LIN {X 0,Y 305.638,Z 167.911,A -85,B 0,C 180,E1 -15829.4,E2 -15829.4} C_VEL
LIN {X 0,Y 305.807,Z 167.885,A -85,B 0,C 180,E1 -15832.074,E2 -15832.074} C_VEL
LIN {X 0,Y 305.686,Z 167.907,A -85,B 0,C 180,E1 -15834.723,E2 -15834.723} C_VEL
LIN {X 0,Y 305.955,Z 167.869,A -85,B 0,C 180,E1 -15838.684,E2 -15838.684} C_VEL
LIN {X 0,Y 305.957,Z 167.872,A -85,B 0,C 180,E1 -15841.316,E2 -15841.316} C_VEL
LIN {X 0,Y 305.845,Z 167.883,A -85,B 0,C 180,E1 -15846.598,E2 -15846.598} C_VEL
LIN {X 0,Y 305.735,Z 167.899,A -85,B 0,C 180,E1 -15849.26,E2 -15849.26} C_VEL
LIN {X 0,Y 305.588,Z 167.911,A -85,B 0,C 180,E1 -15853.296,E2 -15853.296} C_VEL
LIN {X 0,Y 305.593,Z 167.918,A -85,B 0,C 180,E1 -15856.02,E2 -15856.02} C_VEL
LIN {X 0,Y 305.56,Z 167.916,A -85,B 0,C 180,E1 -15859.436,E2 -15859.436} C_VEL
LIN {X 0,Y 305.485,Z 167.93,A -85,B 0,C 180,E1 -15863.039,E2 -15863.039} C_VEL
LIN {X 0,Y 305.546,Z 167.925,A -85,B 0,C 180,E1 -15866.227,E2 -15866.227} C_VEL
LIN {X 0,Y 305.487,Z 167.929,A -85,B 0,C 180,E1 -15869.047,E2 -15869.047} C_VEL
LIN {X 0,Y 305.443,Z 167.94,A -85,B 0,C 180,E1 -15871.952,E2 -15871.952} C_VEL
LIN {X 0,Y 305.462,Z 167.931,A -85,B 0,C 180,E1 -15875.113,E2 -15875.113} C_VEL
LIN {X 0,Y 305.439,Z 167.934,A -85,B 0,C 180,E1 -15878.527,E2 -15878.527} C_VEL
LIN {X 0,Y 305.454,Z 167.934,A -85,B 0,C 180,E1 -15882.586,E2 -15882.586} C_VEL
LIN {X 0,Y 305.421,Z 167.938,A -85,B 0,C 180,E1 -15886.344,E2 -15886.344} C_VEL
LIN {X 0,Y 305.409,Z 167.941,A -85,B 0,C 180,E1 -15889.885,E2 -15889.885} C_VEL
LIN {X 0,Y 305.479,Z 167.934,A -85,B 0,C 180,E1 -15893.633,E2 -15893.633} C_VEL
LIN {X 0,Y 305.508,Z 167.974,A -85,B 0,C 180,E1 -15896.982,E2 -15896.982} C_VEL
LIN {X 0,Y 307.705,Z 177.752,A -85,B 0,C 180,E1 -15900.218,E2 -15900.218} C_VEL
LIN {X 0,Y 309.879,Z 188.802,A -85,B 0,C 180,E1 -15903.685,E2 -15903.685} C_VEL
LIN {X 0,Y 311.303,Z 192.906,A -85,B 0,C 180,E1 -15903.964,E2 -15903.964} C_VEL
LIN {X 0,Y 315.786,Z 216.896,A -85,B 0,C 180,E1 -15904.949,E2 -15904.949} C_VEL
LIN {X 0,Y 317.76,Z 229.786,A -85,B 0,C 180,E1 -15905.428,E2 -15905.428} C_VEL
LIN {X 0,Y 316.105,Z 297.454,A -85,B 0,C 180,E1 -15906.973,E2 -15906.973} C_VEL
LIN {X 0,Y 315.2,Z 310.618,A -85,B 0,C 180,E1 -15907.51,E2 -15907.51} C_VEL
LIN {X 0,Y 314.151,Z 322.724,A -85,B 0,C 180,E1 -15908.252,E2 -15908.252} C_VEL
LIN {X 0,Y 312.759,Z 334.943,A -85,B 0,C 180,E1 -15909.273,E2 -15909.273} C_VEL
LIN {X 0,Y 311.132,Z 346.512,A -85,B 0,C 180,E1 -15910.538,E2 -15910.538} C_VEL
LIN {X 0,Y 309.594,Z 356.932,A -85,B 0,C 180,E1 -15911.983,E2 -15911.983} C_VEL
LIN {X 0,Y 308.215,Z 366.424,A -85,B 0,C 180,E1 -15913.633,E2 -15913.633} C_VEL
LIN {X 0,Y 306.873,Z 374.691,A -85,B 0,C 180,E1 -15915.409,E2 -15915.409} C_VEL
LIN {X 0,Y 305.599,Z 382.114,A -85,B 0,C 180,E1 -15917.381,E2 -15917.381} C_VEL
LIN {X 0,Y 304.716,Z 388.078,A -85,B 0,C 180,E1 -15919.367,E2 -15919.367} C_VEL
LIN {X 0,Y 304.12,Z 392.792,A -85,B 0,C 180,E1 -15921.361,E2 -15921.361} C_VEL
LIN {X 0,Y 303.74,Z 396.394,A -85,B 0,C 180,E1 -15923.357,E2 -15923.357} C_VEL
LIN {X 0,Y 303.618,Z 398.252,A -85,B 0,C 180,E1 -15924.687,E2 -15924.687} C_VEL
LIN {X 0,Y 303.587,Z 399.647,A -85,B 0,C 180,E1 -15926.018,E2 -15926.018} C_VEL
LIN {X 0,Y 303.598,Z 400.642,A -85,B 0,C 180,E1 -15927.346,E2 -15927.346} C_VEL
LIN {X 0,Y 303.556,Z 401.248,A -85,B 0,C 180,E1 -15928.673,E2 -15928.673} C_VEL
LIN {X 0,Y 303.565,Z 401.461,A -85,B 0,C 180,E1 -15930,E2 -15930} C_VEL
LIN {X 0,Y 303.556,Z 401.24,A -85,B 0,C 180,E1 -15931.327,E2 -15931.327} C_VEL
LIN {X 0,Y 303.598,Z 400.63,A -85,B 0,C 180,E1 -15932.654,E2 -15932.654} C_VEL
LIN {X 0,Y 303.588,Z 399.63,A -85,B 0,C 180,E1 -15933.982,E2 -15933.982} C_VEL
LIN {X 0,Y 303.618,Z 397.941,A -85,B 0,C 180,E1 -15935.53,E2 -15935.53} C_VEL
LIN {X 0,Y 303.958,Z 394.057,A -85,B 0,C 180,E1 -15937.974,E2 -15937.974} C_VEL
LIN {X 0,Y 304.472,Z 389.713,A -85,B 0,C 180,E1 -15939.969,E2 -15939.969} C_VEL
LIN {X 0,Y 305.231,Z 384.18,A -85,B 0,C 180,E1 -15941.96,E2 -15941.96} C_VEL
LIN {X 0,Y 306.397,Z 377.279,A -85,B 0,C 180,E1 -15943.936,E2 -15943.936} C_VEL
LIN {X 0,Y 307.521,Z 370.231,A -85,B 0,C 180,E1 -15945.577,E2 -15945.577} C_VEL
LIN {X 0,Y 308.797,Z 361.735,A -85,B 0,C 180,E1 -15947.21,E2 -15947.21} C_VEL
LIN {X 0,Y 310.369,Z 351.24,A -85,B 0,C 180,E1 -15948.825,E2 -15948.825} C_VEL
LIN {X 0,Y 312.149,Z 339.43,A -85,B 0,C 180,E1 -15950.253,E2 -15950.253} C_VEL
LIN {X 0,Y 313.536,Z 327.532,A -85,B 0,C 180,E1 -15951.361,E2 -15951.361} C_VEL
LIN {X 0,Y 314.818,Z 315.152,A -85,B 0,C 180,E1 -15952.217,E2 -15952.217} C_VEL
LIN {X 0,Y 315.848,Z 302.407,A -85,B 0,C 180,E1 -15952.83,E2 -15952.83} C_VEL
LIN {X 0,Y 316.401,Z 288.944,A -85,B 0,C 180,E1 -15953.22,E2 -15953.22} C_VEL
LIN {X 0,Y 317.6,Z 229.007,A -85,B 0,C 180,E1 -15954.578,E2 -15954.578} C_VEL
LIN {X 0,Y 313.198,Z 202.348,A -85,B 0,C 180,E1 -15955.605,E2 -15955.605} C_VEL
LIN {X 0,Y 311.081,Z 192.208,A -85,B 0,C 180,E1 -15956.045,E2 -15956.045} C_VEL
LIN {X 0,Y 309.905,Z 188.891,A -85,B 0,C 180,E1 -15956.258,E2 -15956.258} C_VEL
LIN {X 0,Y 307.676,Z 177.689,A -85,B 0,C 180,E1 -15959.772,E2 -15959.772} C_VEL
LIN {X 0,Y 305.494,Z 167.931,A -85,B 0,C 180,E1 -15963.02,E2 -15963.02} C_VEL
LIN {X 0,Y 305.469,Z 167.937,A -85,B 0,C 180,E1 -15966.74,E2 -15966.74} C_VEL
LIN {X 0,Y 305.409,Z 167.944,A -85,B 0,C 180,E1 -15970.59,E2 -15970.59} C_VEL
LIN {X 0,Y 305.421,Z 167.939,A -85,B 0,C 180,E1 -15973.656,E2 -15973.656} C_VEL
LIN {X 0,Y 305.454,Z 167.934,A -85,B 0,C 180,E1 -15977.414,E2 -15977.414} C_VEL
LIN {X 0,Y 305.467,Z 167.933,A -85,B 0,C 180,E1 -15981.596,E2 -15981.596} C_VEL
LIN {X 0,Y 305.462,Z 167.934,A -85,B 0,C 180,E1 -15984.887,E2 -15984.887} C_VEL
LIN {X 0,Y 305.441,Z 167.939,A -85,B 0,C 180,E1 -15988.358,E2 -15988.358} C_VEL
LIN {X 0,Y 305.486,Z 167.93,A -85,B 0,C 180,E1 -15991.11,E2 -15991.11} C_VEL
LIN {X 0,Y 305.505,Z 167.932,A -85,B 0,C 180,E1 -15994.082,E2 -15994.082} C_VEL
LIN {X 0,Y 305.481,Z 167.931,A -85,B 0,C 180,E1 -15998.401,E2 -15998.401} C_VEL
LIN {X 0,Y 305.579,Z 167.919,A -85,B 0,C 180,E1 -16001.217,E2 -16001.217} C_VEL
LIN {X 0,Y 305.649,Z 167.912,A -85,B 0,C 180,E1 -16005.349,E2 -16005.349} C_VEL
LIN {X 0,Y 305.635,Z 167.913,A -85,B 0,C 180,E1 -16009.4,E2 -16009.4} C_VEL
LIN {X 0,Y 305.796,Z 167.89,A -85,B 0,C 180,E1 -16012.074,E2 -16012.074} C_VEL
LIN {X 0,Y 305.686,Z 167.903,A -85,B 0,C 180,E1 -16014.723,E2 -16014.723} C_VEL
LIN {X 0,Y 305.957,Z 167.87,A -85,B 0,C 180,E1 -16018.684,E2 -16018.684} C_VEL
LIN {X 0,Y 305.956,Z 167.875,A -85,B 0,C 180,E1 -16021.316,E2 -16021.316} C_VEL
LIN {X 0,Y 305.683,Z 167.904,A -85,B 0,C 180,E1 -16025.277,E2 -16025.277} C_VEL
LIN {X 0,Y 305.8,Z 167.891,A -85,B 0,C 180,E1 -16027.926,E2 -16027.926} C_VEL
LIN {X 0,Y 305.603,Z 167.911,A -85,B 0,C 180,E1 -16031.945,E2 -16031.945} C_VEL
LIN {X 0,Y 305.638,Z 167.913,A -85,B 0,C 180,E1 -16035.035,E2 -16035.035} C_VEL
LIN {X 0,Y 305.577,Z 167.919,A -85,B 0,C 180,E1 -16039.445,E2 -16039.445} C_VEL
LIN {X 0,Y 305.491,Z 167.929,A -85,B 0,C 180,E1 -16043.041,E2 -16043.041} C_VEL
LIN {X 0,Y 305.548,Z 167.925,A -85,B 0,C 180,E1 -16046.227,E2 -16046.227} C_VEL
LIN {X 0,Y 305.496,Z 167.929,A -85,B 0,C 180,E1 -16049.05,E2 -16049.05} C_VEL
LIN {X 0,Y 305.465,Z 167.933,A -85,B 0,C 180,E1 -16053.517,E2 -16053.517} C_VEL
LIN {X 0,Y 305.496,Z 167.93,A -85,B 0,C 180,E1 -16056.737,E2 -16056.737} C_VEL
LIN {X 0,Y 305.455,Z 167.935,A -85,B 0,C 180,E1 -16060.6,E2 -16060.6} C_VEL
LIN {X 0,Y 305.426,Z 167.939,A -85,B 0,C 180,E1 -16063.655,E2 -16063.655} C_VEL
LIN {X 0,Y 305.456,Z 167.936,A -85,B 0,C 180,E1 -16067.414,E2 -16067.414} C_VEL
LIN {X 0,Y 305.496,Z 167.934,A -85,B 0,C 180,E1 -16071.601,E2 -16071.601} C_VEL
LIN {X 0,Y 305.463,Z 167.936,A -85,B 0,C 180,E1 -16074.887,E2 -16074.887} C_VEL
LIN {X 0,Y 305.454,Z 167.939,A -85,B 0,C 180,E1 -16078.355,E2 -16078.355} C_VEL
LIN {X 0,Y 305.516,Z 168.02,A -85,B 0,C 180,E1 -16080.66,E2 -16080.66} C_VEL
LIN {X 0,Y 307.507,Z 176.563,A -85,B 0,C 180,E1 -16083.596,E2 -16083.596} C_VEL
LIN {X 0,Y 315.667,Z 197.032,A -85,B 0,C 180,E1 -16084.843,E2 -16084.843} C_VEL
LIN {X 0,Y 318.183,Z 210.063,A -85,B 0,C 180,E1 -16085.375,E2 -16085.375} C_VEL
LIN {X 0,Y 316.488,Z 281.965,A -85,B 0,C 180,E1 -16087.003,E2 -16087.003} C_VEL
LIN {X 0,Y 315.776,Z 294.511,A -85,B 0,C 180,E1 -16087.466,E2 -16087.466} C_VEL
LIN {X 0,Y 314.823,Z 307.319,A -85,B 0,C 180,E1 -16088.215,E2 -16088.215} C_VEL
LIN {X 0,Y 313.582,Z 319.174,A -85,B 0,C 180,E1 -16089.158,E2 -16089.158} C_VEL
LIN {X 0,Y 312.246,Z 329.93,A -85,B 0,C 180,E1 -16090.268,E2 -16090.268} C_VEL
LIN {X 0,Y 310.904,Z 339.817,A -85,B 0,C 180,E1 -16091.55,E2 -16091.55} C_VEL
LIN {X 0,Y 309.587,Z 349.789,A -85,B 0,C 180,E1 -16093.176,E2 -16093.176} C_VEL
LIN {X 0,Y 307.848,Z 359.441,A -85,B 0,C 180,E1 -16095.118,E2 -16095.118} C_VEL
LIN {X 0,Y 306.584,Z 367.133,A -85,B 0,C 180,E1 -16097.085,E2 -16097.085} C_VEL
LIN {X 0,Y 305.376,Z 374.195,A -85,B 0,C 180,E1 -16099.39,E2 -16099.39} C_VEL
LIN {X 0,Y 304.616,Z 378.898,A -85,B 0,C 180,E1 -16101.375,E2 -16101.375} C_VEL
LIN {X 0,Y 304.193,Z 382.623,A -85,B 0,C 180,E1 -16103.447,E2 -16103.447} C_VEL
LIN {X 0,Y 303.977,Z 384.353,A -85,B 0,C 180,E1 -16104.694,E2 -16104.694} C_VEL
LIN {X 0,Y 303.829,Z 385.751,A -85,B 0,C 180,E1 -16106.021,E2 -16106.021} C_VEL
LIN {X 0,Y 303.599,Z 387.359,A -85,B 0,C 180,E1 -16108.673,E2 -16108.673} C_VEL
LIN {X 0,Y 303.571,Z 387.591,A -85,B 0,C 180,E1 -16110,E2 -16110} C_VEL
LIN {X 0,Y 303.599,Z 387.399,A -85,B 0,C 180,E1 -16111.326,E2 -16111.326} C_VEL
LIN {X 0,Y 303.824,Z 385.843,A -85,B 0,C 180,E1 -16113.979,E2 -16113.979} C_VEL
LIN {X 0,Y 304.072,Z 383.108,A -85,B 0,C 180,E1 -16116.352,E2 -16116.352} C_VEL
LIN {X 0,Y 304.609,Z 379.14,A -85,B 0,C 180,E1 -16118.625,E2 -16118.625} C_VEL
LIN {X 0,Y 305.326,Z 374.503,A -85,B 0,C 180,E1 -16120.611,E2 -16120.611} C_VEL
LIN {X 0,Y 306.546,Z 367.51,A -85,B 0,C 180,E1 -16122.917,E2 -16122.917} C_VEL
LIN {X 0,Y 307.809,Z 359.932,A -85,B 0,C 180,E1 -16124.884,E2 -16124.884} C_VEL
LIN {X 0,Y 309.47,Z 350.391,A -85,B 0,C 180,E1 -16126.831,E2 -16126.831} C_VEL
LIN {X 0,Y 310.855,Z 340.545,A -85,B 0,C 180,E1 -16128.452,E2 -16128.452} C_VEL
LIN {X 0,Y 312.384,Z 329.463,A -85,B 0,C 180,E1 -16129.894,E2 -16129.894} C_VEL
LIN {X 0,Y 313.696,Z 318.596,A -85,B 0,C 180,E1 -16131.006,E2 -16131.006} C_VEL
LIN {X 0,Y 314.952,Z 306.588,A -85,B 0,C 180,E1 -16131.948,E2 -16131.948} C_VEL
LIN {X 0,Y 315.811,Z 294.258,A -85,B 0,C 180,E1 -16132.66,E2 -16132.66} C_VEL
LIN {X 0,Y 316.523,Z 281.49,A -85,B 0,C 180,E1 -16133.124,E2 -16133.124} C_VEL
LIN {X 0,Y 318.178,Z 209.471,A -85,B 0,C 180,E1 -16134.756,E2 -16134.756} C_VEL
LIN {X 0,Y 315.6,Z 196.757,A -85,B 0,C 180,E1 -16135.286,E2 -16135.286} C_VEL
LIN {X 0,Y 307.516,Z 176.537,A -85,B 0,C 180,E1 -16136.531,E2 -16136.531} C_VEL
LIN {X 0,Y 305.516,Z 167.929,A -85,B 0,C 180,E1 -16139.569,E2 -16139.569} C_VEL
LIN {X 0,Y 305.465,Z 167.933,A -85,B 0,C 180,E1 -16144.078,E2 -16144.078} C_VEL
LIN {X 0,Y 305.476,Z 167.933,A -85,B 0,C 180,E1 -16146.739,E2 -16146.739} C_VEL
LIN {X 0,Y 305.455,Z 167.937,A -85,B 0,C 180,E1 -16150.599,E2 -16150.599} C_VEL
LIN {X 0,Y 305.426,Z 167.939,A -85,B 0,C 180,E1 -16153.655,E2 -16153.655} C_VEL
LIN {X 0,Y 305.391,Z 167.941,A -85,B 0,C 180,E1 -16154.76,E2 -16154.76} C_VEL
LIN {X 0,Y 304.72,Z 168.029,A -85,B 0,C 180,E1 -16155.86,E2 -16155.86} C_VEL
LIN {X 0,Y 301.893,Z 168.379,A -85,B 0,C 180,E1 -16157.653,E2 -16157.653} C_VEL
LIN {X 0,Y 299.507,Z 168.678,A -85,B 0,C 180,E1 -16159.107,E2 -16159.107} C_VEL
LIN {X 0,Y 298.488,Z 168.804,A -85,B 0,C 180,E1 -16160.233,E2 -16160.233} C_VEL
LIN {X 0,Y 298.408,Z 168.811,A -85,B 0,C 180,E1 -16160.614,E2 -16160.614} C_VEL
LIN {X 0,Y 298.42,Z 168.813,A -85,B 0,C 180,E1 -16163.93,E2 -16163.93} C_VEL
LIN {X 0,Y 298.395,Z 168.816,A -85,B 0,C 180,E1 -16167.983,E2 -16167.983} C_VEL
LIN {X 0,Y 298.463,Z 168.803,A -85,B 0,C 180,E1 -16171.904,E2 -16171.904} C_VEL
LIN {X 0,Y 298.485,Z 168.803,A -85,B 0,C 180,E1 -16174.924,E2 -16174.924} C_VEL
LIN {X 0,Y 298.45,Z 168.806,A -85,B 0,C 180,E1 -16179.315,E2 -16179.315} C_VEL
LIN {X 0,Y 298.538,Z 168.795,A -85,B 0,C 180,E1 -16182.179,E2 -16182.179} C_VEL
LIN {X 0,Y 298.593,Z 168.784,A -85,B 0,C 180,E1 -16184.995,E2 -16184.995} C_VEL
LIN {X 0,Y 298.593,Z 168.791,A -85,B 0,C 180,E1 -16189.147,E2 -16189.147} C_VEL
LIN {X 0,Y 298.754,Z 168.763,A -85,B 0,C 180,E1 -16191.886,E2 -16191.886} C_VEL
LIN {X 0,Y 298.657,Z 168.782,A -85,B 0,C 180,E1 -16194.599,E2 -16194.599} C_VEL
LIN {X 0,Y 298.922,Z 168.744,A -85,B 0,C 180,E1 -16198.653,E2 -16198.653} C_VEL
LIN {X 0,Y 298.923,Z 168.748,A -85,B 0,C 180,E1 -16201.347,E2 -16201.347} C_VEL
LIN {X 0,Y 298.791,Z 168.762,A -85,B 0,C 180,E1 -16206.754,E2 -16206.754} C_VEL
LIN {X 0,Y 298.68,Z 168.778,A -85,B 0,C 180,E1 -16209.48,E2 -16209.48} C_VEL
LIN {X 0,Y 298.551,Z 168.787,A -85,B 0,C 180,E1 -16213.615,E2 -16213.615} C_VEL
LIN {X 0,Y 298.548,Z 168.798,A -85,B 0,C 180,E1 -16216.409,E2 -16216.409} C_VEL
LIN {X 0,Y 298.497,Z 168.796,A -85,B 0,C 180,E1 -16219.647,E2 -16219.647} C_VEL
LIN {X 0,Y 298.428,Z 168.81,A -85,B 0,C 180,E1 -16223.6,E2 -16223.6} C_VEL
LIN {X 0,Y 298.488,Z 168.802,A -85,B 0,C 180,E1 -16226.575,E2 -16226.575} C_VEL
LIN {X 0,Y 298.416,Z 168.812,A -85,B 0,C 180,E1 -16229.642,E2 -16229.642} C_VEL
LIN {X 0,Y 298.395,Z 168.814,A -85,B 0,C 180,E1 -16232.8,E2 -16232.8} C_VEL
LIN {X 0,Y 298.443,Z 168.808,A -85,B 0,C 180,E1 -16236.807,E2 -16236.807} C_VEL
LIN {X 0,Y 298.386,Z 168.816,A -85,B 0,C 180,E1 -16241.088,E2 -16241.088} C_VEL
LIN {X 0,Y 298.398,Z 168.815,A -85,B 0,C 180,E1 -16243.104,E2 -16243.104} C_VEL
LIN {X 0,Y 298.371,Z 168.818,A -85,B 0,C 180,E1 -16246.915,E2 -16246.915} C_VEL
LIN {X 0,Y 298.384,Z 168.817,A -85,B 0,C 180,E1 -16251.011,E2 -16251.011} C_VEL
LIN {X 0,Y 298.417,Z 168.812,A -85,B 0,C 180,E1 -16253.93,E2 -16253.93} C_VEL
LIN {X 0,Y 298.439,Z 168.887,A -85,B 0,C 180,E1 -16256.45,E2 -16256.45} C_VEL
LIN {X 0,Y 300.885,Z 179.606,A -85,B 0,C 180,E1 -16260.1,E2 -16260.1} C_VEL
LIN {X 0,Y 302.697,Z 188.89,A -85,B 0,C 180,E1 -16263.066,E2 -16263.066} C_VEL
LIN {X 0,Y 305.487,Z 196.454,A -85,B 0,C 180,E1 -16263.524,E2 -16263.524} C_VEL
LIN {X 0,Y 310.097,Z 222.353,A -85,B 0,C 180,E1 -16264.597,E2 -16264.597} C_VEL
LIN {X 0,Y 311.306,Z 231.348,A -85,B 0,C 180,E1 -16264.926,E2 -16264.926} C_VEL
LIN {X 0,Y 309.592,Z 297.306,A -85,B 0,C 180,E1 -16266.46,E2 -16266.46} C_VEL
LIN {X 0,Y 308.656,Z 310.465,A -85,B 0,C 180,E1 -16267.006,E2 -16267.006} C_VEL
LIN {X 0,Y 307.573,Z 322.568,A -85,B 0,C 180,E1 -16267.762,E2 -16267.762} C_VEL
LIN {X 0,Y 306.131,Z 334.786,A -85,B 0,C 180,E1 -16268.803,E2 -16268.803} C_VEL
LIN {X 0,Y 304.453,Z 346.353,A -85,B 0,C 180,E1 -16270.093,E2 -16270.093} C_VEL
LIN {X 0,Y 302.809,Z 356.772,A -85,B 0,C 180,E1 -16271.565,E2 -16271.565} C_VEL
LIN {X 0,Y 301.55,Z 365.173,A -85,B 0,C 180,E1 -16273.039,E2 -16273.039} C_VEL
LIN {X 0,Y 300.249,Z 373.156,A -85,B 0,C 180,E1 -16274.732,E2 -16274.732} C_VEL
LIN {X 0,Y 298.834,Z 380.832,A -85,B 0,C 180,E1 -16276.744,E2 -16276.744} C_VEL
LIN {X 0,Y 297.719,Z 387.917,A -85,B 0,C 180,E1 -16279.114,E2 -16279.114} C_VEL
LIN {X 0,Y 297.069,Z 392.63,A -85,B 0,C 180,E1 -16281.154,E2 -16281.154} C_VEL
LIN {X 0,Y 296.687,Z 396.233,A -85,B 0,C 180,E1 -16283.198,E2 -16283.198} C_VEL
LIN {X 0,Y 296.532,Z 398.09,A -85,B 0,C 180,E1 -16284.56,E2 -16284.56} C_VEL
LIN {X 0,Y 296.488,Z 399.484,A -85,B 0,C 180,E1 -16285.922,E2 -16285.922} C_VEL
LIN {X 0,Y 296.522,Z 400.481,A -85,B 0,C 180,E1 -16287.283,E2 -16287.283} C_VEL
LIN {X 0,Y 296.476,Z 401.086,A -85,B 0,C 180,E1 -16288.642,E2 -16288.642} C_VEL
LIN {X 0,Y 296.482,Z 401.299,A -85,B 0,C 180,E1 -16290,E2 -16290} C_VEL
LIN {X 0,Y 296.476,Z 401.078,A -85,B 0,C 180,E1 -16291.358,E2 -16291.358} C_VEL
LIN {X 0,Y 296.522,Z 400.468,A -85,B 0,C 180,E1 -16292.717,E2 -16292.717} C_VEL
LIN {X 0,Y 296.489,Z 399.467,A -85,B 0,C 180,E1 -16294.078,E2 -16294.078} C_VEL
LIN {X 0,Y 296.546,Z 397.98,A -85,B 0,C 180,E1 -16295.509,E2 -16295.509} C_VEL
LIN {X 0,Y 296.789,Z 395.124,A -85,B 0,C 180,E1 -16297.484,E2 -16297.484} C_VEL
LIN {X 0,Y 297.26,Z 391.145,A -85,B 0,C 180,E1 -16299.526,E2 -16299.526} C_VEL
LIN {X 0,Y 298.12,Z 385.028,A -85,B 0,C 180,E1 -16301.904,E2 -16301.904} C_VEL
LIN {X 0,Y 299.277,Z 378.35,A -85,B 0,C 180,E1 -16303.928,E2 -16303.928} C_VEL
LIN {X 0,Y 300.659,Z 370.066,A -85,B 0,C 180,E1 -16305.942,E2 -16305.942} C_VEL
LIN {X 0,Y 302,Z 361.569,A -85,B 0,C 180,E1 -16307.61,E2 -16307.61} C_VEL
LIN {X 0,Y 303.664,Z 351.074,A -85,B 0,C 180,E1 -16309.257,E2 -16309.257} C_VEL
LIN {X 0,Y 305.484,Z 339.263,A -85,B 0,C 180,E1 -16310.715,E2 -16310.715} C_VEL
LIN {X 0,Y 306.935,Z 327.364,A -85,B 0,C 180,E1 -16311.844,E2 -16311.844} C_VEL
LIN {X 0,Y 308.259,Z 314.982,A -85,B 0,C 180,E1 -16312.716,E2 -16312.716} C_VEL
LIN {X 0,Y 309.327,Z 302.234,A -85,B 0,C 180,E1 -16313.34,E2 -16313.34} C_VEL
LIN {X 0,Y 309.894,Z 288.76,A -85,B 0,C 180,E1 -16313.737,E2 -16313.737} C_VEL
LIN {X 0,Y 311.146,Z 230.104,A -85,B 0,C 180,E1 -16315.091,E2 -16315.091} C_VEL
LIN {X 0,Y 306.959,Z 204.259,A -85,B 0,C 180,E1 -16316.111,E2 -16316.111} C_VEL
LIN {X 0,Y 304.938,Z 194.729,A -85,B 0,C 180,E1 -16316.541,E2 -16316.541} C_VEL
LIN {X 0,Y 302.695,Z 188.746,A -85,B 0,C 180,E1 -16316.922,E2 -16316.922} C_VEL
LIN {X 0,Y 300.479,Z 177.864,A -85,B 0,C 180,E1 -16320.448,E2 -16320.448} C_VEL
LIN {X 0,Y 298.448,Z 168.809,A -85,B 0,C 180,E1 -16323.6,E2 -16323.6} C_VEL
LIN {X 0,Y 298.403,Z 168.814,A -85,B 0,C 180,E1 -16327.76,E2 -16327.76} C_VEL
LIN {X 0,Y 298.348,Z 168.822,A -85,B 0,C 180,E1 -16331.268,E2 -16331.268} C_VEL
LIN {X 0,Y 298.399,Z 168.816,A -85,B 0,C 180,E1 -16333.103,E2 -16333.103} C_VEL
LIN {X 0,Y 298.403,Z 168.814,A -85,B 0,C 180,E1 -16336.921,E2 -16336.921} C_VEL
LIN {X 0,Y 298.398,Z 168.814,A -85,B 0,C 180,E1 -16341.007,E2 -16341.007} C_VEL
LIN {X 0,Y 298.418,Z 168.813,A -85,B 0,C 180,E1 -16343.93,E2 -16343.93} C_VEL
LIN {X 0,Y 298.388,Z 168.818,A -85,B 0,C 180,E1 -16347.985,E2 -16347.985} C_VEL
LIN {X 0,Y 298.422,Z 168.813,A -85,B 0,C 180,E1 -16351.9,E2 -16351.9} C_VEL
LIN {X 0,Y 298.448,Z 168.807,A -85,B 0,C 180,E1 -16354.921,E2 -16354.921} C_VEL
LIN {X 0,Y 298.437,Z 168.809,A -85,B 0,C 180,E1 -16359.314,E2 -16359.314} C_VEL
LIN {X 0,Y 298.534,Z 168.795,A -85,B 0,C 180,E1 -16362.179,E2 -16362.179} C_VEL
LIN {X 0,Y 298.593,Z 168.789,A -85,B 0,C 180,E1 -16364.995,E2 -16364.995} C_VEL
LIN {X 0,Y 298.591,Z 168.788,A -85,B 0,C 180,E1 -16369.147,E2 -16369.147} C_VEL
LIN {X 0,Y 298.741,Z 168.77,A -85,B 0,C 180,E1 -16371.885,E2 -16371.885} C_VEL
LIN {X 0,Y 298.656,Z 168.778,A -85,B 0,C 180,E1 -16374.599,E2 -16374.599} C_VEL
LIN {X 0,Y 298.924,Z 168.746,A -85,B 0,C 180,E1 -16378.653,E2 -16378.653} C_VEL
LIN {X 0,Y 298.922,Z 168.751,A -85,B 0,C 180,E1 -16381.347,E2 -16381.347} C_VEL
LIN {X 0,Y 298.785,Z 168.764,A -85,B 0,C 180,E1 -16386.754,E2 -16386.754} C_VEL
LIN {X 0,Y 298.636,Z 168.784,A -85,B 0,C 180,E1 -16389.482,E2 -16389.482} C_VEL
LIN {X 0,Y 298.552,Z 168.794,A -85,B 0,C 180,E1 -16393.615,E2 -16393.615} C_VEL
LIN {X 0,Y 298.549,Z 168.796,A -85,B 0,C 180,E1 -16396.409,E2 -16396.409} C_VEL
LIN {X 0,Y 298.512,Z 168.799,A -85,B 0,C 180,E1 -16399.655,E2 -16399.655} C_VEL
LIN {X 0,Y 298.458,Z 168.804,A -85,B 0,C 180,E1 -16403.598,E2 -16403.598} C_VEL
LIN {X 0,Y 298.49,Z 168.802,A -85,B 0,C 180,E1 -16406.575,E2 -16406.575} C_VEL
LIN {X 0,Y 298.421,Z 168.81,A -85,B 0,C 180,E1 -16409.641,E2 -16409.641} C_VEL
LIN {X 0,Y 298.396,Z 168.814,A -85,B 0,C 180,E1 -16412.8,E2 -16412.8} C_VEL
LIN {X 0,Y 298.465,Z 168.805,A -85,B 0,C 180,E1 -16416.812,E2 -16416.812} C_VEL
LIN {X 0,Y 298.388,Z 168.815,A -85,B 0,C 180,E1 -16421.088,E2 -16421.088} C_VEL
LIN {X 0,Y 298.399,Z 168.812,A -85,B 0,C 180,E1 -16423.104,E2 -16423.104} C_VEL
LIN {X 0,Y 298.404,Z 168.812,A -85,B 0,C 180,E1 -16426.921,E2 -16426.921} C_VEL
LIN {X 0,Y 298.416,Z 168.812,A -85,B 0,C 180,E1 -16431.004,E2 -16431.004} C_VEL
LIN {X 0,Y 298.42,Z 168.814,A -85,B 0,C 180,E1 -16433.93,E2 -16433.93} C_VEL
LIN {X 0,Y 298.397,Z 168.82,A -85,B 0,C 180,E1 -16437.983,E2 -16437.983} C_VEL
LIN {X 0,Y 298.482,Z 169.011,A -85,B 0,C 180,E1 -16440.172,E2 -16440.172} C_VEL
LIN {X 0,Y 300.305,Z 176.779,A -85,B 0,C 180,E1 -16442.915,E2 -16442.915} C_VEL
LIN {X 0,Y 308.302,Z 196.296,A -85,B 0,C 180,E1 -16444.175,E2 -16444.175} C_VEL
LIN {X 0,Y 309.882,Z 200.941,A -85,B 0,C 180,E1 -16444.434,E2 -16444.434} C_VEL
LIN {X 0,Y 311.73,Z 211.09,A -85,B 0,C 180,E1 -16444.852,E2 -16444.852} C_VEL
LIN {X 0,Y 309.973,Z 282.148,A -85,B 0,C 180,E1 -16446.491,E2 -16446.491} C_VEL
LIN {X 0,Y 309.254,Z 294.683,A -85,B 0,C 180,E1 -16446.964,E2 -16446.964} C_VEL
LIN {X 0,Y 308.247,Z 307.489,A -85,B 0,C 180,E1 -16447.725,E2 -16447.725} C_VEL
LIN {X 0,Y 306.977,Z 319.342,A -85,B 0,C 180,E1 -16448.688,E2 -16448.688} C_VEL
LIN {X 0,Y 305.583,Z 330.097,A -85,B 0,C 180,E1 -16449.819,E2 -16449.819} C_VEL
LIN {X 0,Y 304.176,Z 339.983,A -85,B 0,C 180,E1 -16451.127,E2 -16451.127} C_VEL
LIN {X 0,Y 302.794,Z 349.954,A -85,B 0,C 180,E1 -16452.787,E2 -16452.787} C_VEL
LIN {X 0,Y 301.003,Z 359.605,A -85,B 0,C 180,E1 -16454.771,E2 -16454.771} C_VEL
LIN {X 0,Y 299.661,Z 367.298,A -85,B 0,C 180,E1 -16456.781,E2 -16456.781} C_VEL
LIN {X 0,Y 298.395,Z 374.359,A -85,B 0,C 180,E1 -16459.139,E2 -16459.139} C_VEL
LIN {X 0,Y 297.597,Z 379.061,A -85,B 0,C 180,E1 -16461.17,E2 -16461.17} C_VEL
LIN {X 0,Y 297.107,Z 383.06,A -85,B 0,C 180,E1 -16463.467,E2 -16463.467} C_VEL
LIN {X 0,Y 296.748,Z 385.913,A -85,B 0,C 180,E1 -16465.926,E2 -16465.926} C_VEL
LIN {X 0,Y 296.615,Z 386.908,A -85,B 0,C 180,E1 -16467.284,E2 -16467.284} C_VEL
LIN {X 0,Y 296.488,Z 387.753,A -85,B 0,C 180,E1 -16470,E2 -16470} C_VEL
LIN {X 0,Y 296.519,Z 387.561,A -85,B 0,C 180,E1 -16471.358,E2 -16471.358} C_VEL
LIN {X 0,Y 296.613,Z 386.974,A -85,B 0,C 180,E1 -16472.716,E2 -16472.716} C_VEL
LIN {X 0,Y 296.742,Z 386.005,A -85,B 0,C 180,E1 -16474.074,E2 -16474.074} C_VEL
LIN {X 0,Y 296.998,Z 383.474,A -85,B 0,C 180,E1 -16476.347,E2 -16476.347} C_VEL
LIN {X 0,Y 297.589,Z 379.301,A -85,B 0,C 180,E1 -16478.83,E2 -16478.83} C_VEL
LIN {X 0,Y 298.351,Z 374.664,A -85,B 0,C 180,E1 -16480.862,E2 -16480.862} C_VEL
LIN {X 0,Y 299.618,Z 367.67,A -85,B 0,C 180,E1 -16483.22,E2 -16483.22} C_VEL
LIN {X 0,Y 300.968,Z 360.092,A -85,B 0,C 180,E1 -16485.23,E2 -16485.23} C_VEL
LIN {X 0,Y 302.674,Z 350.55,A -85,B 0,C 180,E1 -16487.22,E2 -16487.22} C_VEL
LIN {X 0,Y 304.121,Z 340.704,A -85,B 0,C 180,E1 -16488.876,E2 -16488.876} C_VEL
LIN {X 0,Y 305.704,Z 329.62,A -85,B 0,C 180,E1 -16490.348,E2 -16490.348} C_VEL
LIN {X 0,Y 307.1,Z 318.752,A -85,B 0,C 180,E1 -16491.479,E2 -16491.479} C_VEL
LIN {X 0,Y 308.385,Z 306.742,A -85,B 0,C 180,E1 -16492.441,E2 -16492.441} C_VEL
LIN {X 0,Y 309.279,Z 294.409,A -85,B 0,C 180,E1 -16493.166,E2 -16493.166} C_VEL
LIN {X 0,Y 310.025,Z 281.631,A -85,B 0,C 180,E1 -16493.638,E2 -16493.638} C_VEL
LIN {X 0,Y 311.68,Z 210.328,A -85,B 0,C 180,E1 -16495.29,E2 -16495.29} C_VEL
LIN {X 0,Y 309.368,Z 198.967,A -85,B 0,C 180,E1 -16495.78,E2 -16495.78} C_VEL
LIN {X 0,Y 301.358,Z 179.337,A -85,B 0,C 180,E1 -16497.037,E2 -16497.037} C_VEL
LIN {X 0,Y 300.321,Z 176.714,A -85,B 0,C 180,E1 -16497.219,E2 -16497.219} C_VEL
LIN {X 0,Y 298.445,Z 168.81,A -85,B 0,C 180,E1 -16500.027,E2 -16500.027} C_VEL
LIN {X 0,Y 298.429,Z 168.807,A -85,B 0,C 180,E1 -16504.487,E2 -16504.487} C_VEL
LIN {X 0,Y 298.414,Z 168.811,A -85,B 0,C 180,E1 -16507.758,E2 -16507.758} C_VEL
LIN {X 0,Y 298.385,Z 168.815,A -85,B 0,C 180,E1 -16511.261,E2 -16511.261} C_VEL
LIN {X 0,Y 298.354,Z 168.817,A -85,B 0,C 180,E1 -16515.035,E2 -16515.035} C_VEL
LIN {X 0,Y 298.384,Z 168.814,A -85,B 0,C 180,E1 -16518.738,E2 -16518.738} C_VEL
LIN {X 0,Y 298.408,Z 168.811,A -85,B 0,C 180,E1 -16520.614,E2 -16520.614} C_VEL
LIN {X 0,Y 297.749,Z 168.894,A -85,B 0,C 180,E1 -16521.74,E2 -16521.74} C_VEL
LIN {X 0,Y 294.904,Z 169.248,A -85,B 0,C 180,E1 -16523.575,E2 -16523.575} C_VEL
LIN {X 0,Y 292.477,Z 169.55,A -85,B 0,C 180,E1 -16525.063,E2 -16525.063} C_VEL
LIN {X 0,Y 291.423,Z 169.679,A -85,B 0,C 180,E1 -16526.216,E2 -16526.216} C_VEL
LIN {X 0,Y 291.331,Z 169.688,A -85,B 0,C 180,E1 -16526.607,E2 -16526.607} C_VEL
LIN {X 0,Y 291.387,Z 169.685,A -85,B 0,C 180,E1 -16530.26,E2 -16530.26} C_VEL
LIN {X 0,Y 291.417,Z 169.683,A -85,B 0,C 180,E1 -16534.272,E2 -16534.272} C_VEL
LIN {X 0,Y 291.381,Z 169.686,A -85,B 0,C 180,E1 -16537.299,E2 -16537.299} C_VEL
LIN {X 0,Y 291.458,Z 169.678,A -85,B 0,C 180,E1 -16540.27,E2 -16540.27} C_VEL
LIN {X 0,Y 291.555,Z 169.659,A -85,B 0,C 180,E1 -16544.624,E2 -16544.624} C_VEL
LIN {X 0,Y 291.536,Z 169.671,A -85,B 0,C 180,E1 -16548.88,E2 -16548.88} C_VEL
LIN {X 0,Y 291.705,Z 169.641,A -85,B 0,C 180,E1 -16551.688,E2 -16551.688} C_VEL
LIN {X 0,Y 291.628,Z 169.657,A -85,B 0,C 180,E1 -16554.468,E2 -16554.468} C_VEL
LIN {X 0,Y 291.888,Z 169.62,A -85,B 0,C 180,E1 -16558.62,E2 -16558.62} C_VEL
LIN {X 0,Y 291.889,Z 169.624,A -85,B 0,C 180,E1 -16561.38,E2 -16561.38} C_VEL
LIN {X 0,Y 291.74,Z 169.64,A -85,B 0,C 180,E1 -16566.918,E2 -16566.918} C_VEL
LIN {X 0,Y 291.629,Z 169.656,A -85,B 0,C 180,E1 -16569.712,E2 -16569.712} C_VEL
LIN {X 0,Y 291.521,Z 169.664,A -85,B 0,C 180,E1 -16573.95,E2 -16573.95} C_VEL
LIN {X 0,Y 291.485,Z 169.674,A -85,B 0,C 180,E1 -16576.818,E2 -16576.818} C_VEL
LIN {X 0,Y 291.45,Z 169.674,A -85,B 0,C 180,E1 -16579.875,E2 -16579.875} C_VEL
LIN {X 0,Y 291.382,Z 169.686,A -85,B 0,C 180,E1 -16584.207,E2 -16584.207} C_VEL
LIN {X 0,Y 291.42,Z 169.682,A -85,B 0,C 180,E1 -16587.272,E2 -16587.272} C_VEL
LIN {X 0,Y 291.334,Z 169.692,A -85,B 0,C 180,E1 -16590.437,E2 -16590.437} C_VEL
LIN {X 0,Y 291.344,Z 169.693,A -85,B 0,C 180,E1 -16593.698,E2 -16593.698} C_VEL
LIN {X 0,Y 291.372,Z 169.69,A -85,B 0,C 180,E1 -16597.253,E2 -16597.253} C_VEL
LIN {X 0,Y 291.331,Z 169.694,A -85,B 0,C 180,E1 -16600.643,E2 -16600.643} C_VEL
LIN {X 0,Y 291.29,Z 169.697,A -85,B 0,C 180,E1 -16604.402,E2 -16604.402} C_VEL
LIN {X 0,Y 291.295,Z 169.698,A -85,B 0,C 180,E1 -16608.412,E2 -16608.412} C_VEL
LIN {X 0,Y 291.335,Z 169.696,A -85,B 0,C 180,E1 -16611.156,E2 -16611.156} C_VEL
LIN {X 0,Y 291.36,Z 169.692,A -85,B 0,C 180,E1 -16614.626,E2 -16614.626} C_VEL
LIN {X 0,Y 291.409,Z 169.842,A -85,B 0,C 180,E1 -16615.907,E2 -16615.907} C_VEL
LIN {X 0,Y 293.746,Z 179.954,A -85,B 0,C 180,E1 -16619.465,E2 -16619.465} C_VEL
LIN {X 0,Y 295.479,Z 188.628,A -85,B 0,C 180,E1 -16622.35,E2 -16622.35} C_VEL
LIN {X 0,Y 299.423,Z 199.198,A -85,B 0,C 180,E1 -16623.021,E2 -16623.021} C_VEL
LIN {X 0,Y 303.691,Z 223.504,A -85,B 0,C 180,E1 -16624.055,E2 -16624.055} C_VEL
LIN {X 0,Y 304.878,Z 231.794,A -85,B 0,C 180,E1 -16624.375,E2 -16624.375} C_VEL
LIN {X 0,Y 303.102,Z 297.157,A -85,B 0,C 180,E1 -16625.924,E2 -16625.924} C_VEL
LIN {X 0,Y 302.145,Z 310.312,A -85,B 0,C 180,E1 -16626.481,E2 -16626.481} C_VEL
LIN {X 0,Y 301.023,Z 322.413,A -85,B 0,C 180,E1 -16627.252,E2 -16627.252} C_VEL
LIN {X 0,Y 299.531,Z 334.628,A -85,B 0,C 180,E1 -16628.312,E2 -16628.312} C_VEL
LIN {X 0,Y 297.781,Z 346.195,A -85,B 0,C 180,E1 -16629.628,E2 -16629.628} C_VEL
LIN {X 0,Y 296.06,Z 356.612,A -85,B 0,C 180,E1 -16631.129,E2 -16631.129} C_VEL
LIN {X 0,Y 294.631,Z 365.694,A -85,B 0,C 180,E1 -16632.768,E2 -16632.768} C_VEL
LIN {X 0,Y 293.09,Z 374.37,A -85,B 0,C 180,E1 -16634.706,E2 -16634.706} C_VEL
LIN {X 0,Y 291.682,Z 381.791,A -85,B 0,C 180,E1 -16636.768,E2 -16636.768} C_VEL
LIN {X 0,Y 290.729,Z 387.756,A -85,B 0,C 180,E1 -16638.849,E2 -16638.849} C_VEL
LIN {X 0,Y 290.036,Z 392.469,A -85,B 0,C 180,E1 -16640.938,E2 -16640.938} C_VEL
LIN {X 0,Y 289.606,Z 396.071,A -85,B 0,C 180,E1 -16643.031,E2 -16643.031} C_VEL
LIN {X 0,Y 289.427,Z 398.127,A -85,B 0,C 180,E1 -16644.612,E2 -16644.612} C_VEL
LIN {X 0,Y 289.426,Z 400.319,A -85,B 0,C 180,E1 -16647.216,E2 -16647.216} C_VEL
LIN {X 0,Y 289.398,Z 400.925,A -85,B 0,C 180,E1 -16648.609,E2 -16648.609} C_VEL
LIN {X 0,Y 289.401,Z 401.137,A -85,B 0,C 180,E1 -16650,E2 -16650} C_VEL
LIN {X 0,Y 289.398,Z 400.917,A -85,B 0,C 180,E1 -16651.392,E2 -16651.392} C_VEL
LIN {X 0,Y 289.426,Z 400.306,A -85,B 0,C 180,E1 -16652.784,E2 -16652.784} C_VEL
LIN {X 0,Y 289.477,Z 397.903,A -85,B 0,C 180,E1 -16655.573,E2 -16655.573} C_VEL
LIN {X 0,Y 289.72,Z 394.96,A -85,B 0,C 180,E1 -16657.667,E2 -16657.667} C_VEL
LIN {X 0,Y 290.243,Z 390.981,A -85,B 0,C 180,E1 -16659.759,E2 -16659.759} C_VEL
LIN {X 0,Y 291.124,Z 384.863,A -85,B 0,C 180,E1 -16662.195,E2 -16662.195} C_VEL
LIN {X 0,Y 292.353,Z 378.186,A -85,B 0,C 180,E1 -16664.265,E2 -16664.265} C_VEL
LIN {X 0,Y 293.82,Z 369.901,A -85,B 0,C 180,E1 -16666.323,E2 -16666.323} C_VEL
LIN {X 0,Y 295.219,Z 361.404,A -85,B 0,C 180,E1 -16668.028,E2 -16668.028} C_VEL
LIN {X 0,Y 296.965,Z 350.909,A -85,B 0,C 180,E1 -16669.709,E2 -16669.709} C_VEL
LIN {X 0,Y 298.6,Z 340.525,A -85,B 0,C 180,E1 -16671.035,E2 -16671.035} C_VEL
LIN {X 0,Y 300.145,Z 329.135,A -85,B 0,C 180,E1 -16672.183,E2 -16672.183} C_VEL
LIN {X 0,Y 301.469,Z 317.415,A -85,B 0,C 180,E1 -16673.075,E2 -16673.075} C_VEL
LIN {X 0,Y 302.609,Z 304.815,A -85,B 0,C 180,E1 -16673.753,E2 -16673.753} C_VEL
LIN {X 0,Y 303.357,Z 291.961,A -85,B 0,C 180,E1 -16674.191,E2 -16674.191} C_VEL
LIN {X 0,Y 304.669,Z 230.39,A -85,B 0,C 180,E1 -16675.65,E2 -16675.65} C_VEL
LIN {X 0,Y 300.629,Z 205.744,A -85,B 0,C 180,E1 -16676.66,E2 -16676.66} C_VEL
LIN {X 0,Y 298.85,Z 197.327,A -85,B 0,C 180,E1 -16677.052,E2 -16677.052} C_VEL
LIN {X 0,Y 295.488,Z 188.49,A -85,B 0,C 180,E1 -16677.656,E2 -16677.656} C_VEL
LIN {X 0,Y 293.107,Z 177.162,A -85,B 0,C 180,E1 -16681.463,E2 -16681.463} C_VEL
LIN {X 0,Y 291.378,Z 169.69,A -85,B 0,C 180,E1 -16684.147,E2 -16684.147} C_VEL
LIN {X 0,Y 291.368,Z 169.692,A -85,B 0,C 180,E1 -16687.252,E2 -16687.252} C_VEL
LIN {X 0,Y 291.3,Z 169.702,A -85,B 0,C 180,E1 -16690.648,E2 -16690.648} C_VEL
LIN {X 0,Y 291.291,Z 169.703,A -85,B 0,C 180,E1 -16694.402,E2 -16694.402} C_VEL
LIN {X 0,Y 291.326,Z 169.699,A -85,B 0,C 180,E1 -16698.404,E2 -16698.404} C_VEL
LIN {X 0,Y 291.347,Z 169.692,A -85,B 0,C 180,E1 -16701.157,E2 -16701.157} C_VEL
LIN {X 0,Y 291.361,Z 169.692,A -85,B 0,C 180,E1 -16704.626,E2 -16704.626} C_VEL
LIN {X 0,Y 291.365,Z 169.692,A -85,B 0,C 180,E1 -16707.95,E2 -16707.95} C_VEL
LIN {X 0,Y 291.351,Z 169.691,A -85,B 0,C 180,E1 -16711.155,E2 -16711.155} C_VEL
LIN {X 0,Y 291.376,Z 169.691,A -85,B 0,C 180,E1 -16714.268,E2 -16714.268} C_VEL
LIN {X 0,Y 291.372,Z 169.686,A -85,B 0,C 180,E1 -16717.299,E2 -16717.299} C_VEL
LIN {X 0,Y 291.458,Z 169.678,A -85,B 0,C 180,E1 -16720.27,E2 -16720.27} C_VEL
LIN {X 0,Y 291.555,Z 169.666,A -85,B 0,C 180,E1 -16724.624,E2 -16724.624} C_VEL
LIN {X 0,Y 291.535,Z 169.666,A -85,B 0,C 180,E1 -16728.881,E2 -16728.881} C_VEL
LIN {X 0,Y 291.688,Z 169.65,A -85,B 0,C 180,E1 -16731.688,E2 -16731.688} C_VEL
LIN {X 0,Y 291.627,Z 169.654,A -85,B 0,C 180,E1 -16734.468,E2 -16734.468} C_VEL
LIN {X 0,Y 291.89,Z 169.622,A -85,B 0,C 180,E1 -16738.62,E2 -16738.62} C_VEL
LIN {X 0,Y 291.889,Z 169.627,A -85,B 0,C 180,E1 -16741.38,E2 -16741.38} C_VEL
LIN {X 0,Y 291.734,Z 169.643,A -85,B 0,C 180,E1 -16746.918,E2 -16746.918} C_VEL
LIN {X 0,Y 291.575,Z 169.662,A -85,B 0,C 180,E1 -16749.714,E2 -16749.714} C_VEL
LIN {X 0,Y 291.522,Z 169.669,A -85,B 0,C 180,E1 -16753.95,E2 -16753.95} C_VEL
LIN {X 0,Y 291.487,Z 169.673,A -85,B 0,C 180,E1 -16756.818,E2 -16756.818} C_VEL
LIN {X 0,Y 291.451,Z 169.679,A -85,B 0,C 180,E1 -16759.875,E2 -16759.875} C_VEL
LIN {X 0,Y 291.401,Z 169.685,A -85,B 0,C 180,E1 -16764.205,E2 -16764.205} C_VEL
LIN {X 0,Y 291.423,Z 169.678,A -85,B 0,C 180,E1 -16767.272,E2 -16767.272} C_VEL
LIN {X 0,Y 291.338,Z 169.695,A -85,B 0,C 180,E1 -16770.437,E2 -16770.437} C_VEL
LIN {X 0,Y 291.345,Z 169.692,A -85,B 0,C 180,E1 -16773.699,E2 -16773.699} C_VEL
LIN {X 0,Y 291.394,Z 169.686,A -85,B 0,C 180,E1 -16777.259,E2 -16777.259} C_VEL
LIN {X 0,Y 291.334,Z 169.694,A -85,B 0,C 180,E1 -16780.643,E2 -16780.643} C_VEL
LIN {X 0,Y 291.291,Z 169.699,A -85,B 0,C 180,E1 -16784.402,E2 -16784.402} C_VEL
LIN {X 0,Y 291.327,Z 169.695,A -85,B 0,C 180,E1 -16788.405,E2 -16788.405} C_VEL
LIN {X 0,Y 291.365,Z 169.691,A -85,B 0,C 180,E1 -16791.16,E2 -16791.16} C_VEL
LIN {X 0,Y 291.362,Z 169.693,A -85,B 0,C 180,E1 -16794.626,E2 -16794.626} C_VEL
LIN {X 0,Y 291.378,Z 169.69,A -85,B 0,C 180,E1 -16799.166,E2 -16799.166} C_VEL
LIN {X 0,Y 291.396,Z 169.768,A -85,B 0,C 180,E1 -16799.57,E2 -16799.57} C_VEL
LIN {X 0,Y 293.154,Z 177.108,A -85,B 0,C 180,E1 -16802.201,E2 -16802.201} C_VEL
LIN {X 0,Y 301.277,Z 196.292,A -85,B 0,C 180,E1 -16803.521,E2 -16803.521} C_VEL
LIN {X 0,Y 303.752,Z 203.42,A -85,B 0,C 180,E1 -16803.939,E2 -16803.939} C_VEL
LIN {X 0,Y 305.324,Z 211.89,A -85,B 0,C 180,E1 -16804.302,E2 -16804.302} C_VEL
LIN {X 0,Y 303.5,Z 282.33,A -85,B 0,C 180,E1 -16805.958,E2 -16805.958} C_VEL
LIN {X 0,Y 302.755,Z 294.856,A -85,B 0,C 180,E1 -16806.44,E2 -16806.44} C_VEL
LIN {X 0,Y 301.7,Z 307.658,A -85,B 0,C 180,E1 -16807.215,E2 -16807.215} C_VEL
LIN {X 0,Y 300.381,Z 319.51,A -85,B 0,C 180,E1 -16808.196,E2 -16808.196} C_VEL
LIN {X 0,Y 298.949,Z 330.263,A -85,B 0,C 180,E1 -16809.351,E2 -16809.351} C_VEL
LIN {X 0,Y 297.446,Z 340.15,A -85,B 0,C 180,E1 -16810.683,E2 -16810.683} C_VEL
LIN {X 0,Y 296.011,Z 350.12,A -85,B 0,C 180,E1 -16812.379,E2 -16812.379} C_VEL
LIN {X 0,Y 294.167,Z 359.77,A -85,B 0,C 180,E1 -16814.409,E2 -16814.409} C_VEL
LIN {X 0,Y 292.719,Z 367.463,A -85,B 0,C 180,E1 -16816.462,E2 -16816.462} C_VEL
LIN {X 0,Y 291.425,Z 374.523,A -85,B 0,C 180,E1 -16818.876,E2 -16818.876} C_VEL
LIN {X 0,Y 290.575,Z 379.225,A -85,B 0,C 180,E1 -16820.955,E2 -16820.955} C_VEL
LIN {X 0,Y 290.015,Z 383.486,A -85,B 0,C 180,E1 -16823.497,E2 -16823.497} C_VEL
LIN {X 0,Y 289.67,Z 386.076,A -85,B 0,C 180,E1 -16825.826,E2 -16825.826} C_VEL
LIN {X 0,Y 289.545,Z 387.07,A -85,B 0,C 180,E1 -16827.217,E2 -16827.217} C_VEL
LIN {X 0,Y 289.408,Z 387.914,A -85,B 0,C 180,E1 -16830,E2 -16830} C_VEL
LIN {X 0,Y 289.441,Z 387.722,A -85,B 0,C 180,E1 -16831.391,E2 -16831.391} C_VEL
LIN {X 0,Y 289.544,Z 387.135,A -85,B 0,C 180,E1 -16832.782,E2 -16832.782} C_VEL
LIN {X 0,Y 289.664,Z 386.166,A -85,B 0,C 180,E1 -16834.174,E2 -16834.174} C_VEL
LIN {X 0,Y 289.907,Z 383.876,A -85,B 0,C 180,E1 -16836.313,E2 -16836.313} C_VEL
LIN {X 0,Y 290.377,Z 380.743,A -85,B 0,C 180,E1 -16838.35,E2 -16838.35} C_VEL
LIN {X 0,Y 291.08,Z 376.487,A -85,B 0,C 180,E1 -16840.433,E2 -16840.433} C_VEL
LIN {X 0,Y 292.278,Z 370.04,A -85,B 0,C 180,E1 -16842.851,E2 -16842.851} C_VEL
LIN {X 0,Y 293.541,Z 362.957,A -85,B 0,C 180,E1 -16844.914,E2 -16844.914} C_VEL
LIN {X 0,Y 295.304,Z 354.126,A -85,B 0,C 180,E1 -16846.95,E2 -16846.95} C_VEL
LIN {X 0,Y 296.81,Z 344.687,A -85,B 0,C 180,E1 -16848.712,E2 -16848.712} C_VEL
LIN {X 0,Y 298.478,Z 333.747,A -85,B 0,C 180,E1 -16850.322,E2 -16850.322} C_VEL
LIN {X 0,Y 300.096,Z 322.293,A -85,B 0,C 180,E1 -16851.645,E2 -16851.645} C_VEL
LIN {X 0,Y 301.557,Z 310.279,A -85,B 0,C 180,E1 -16852.706,E2 -16852.706} C_VEL
LIN {X 0,Y 302.614,Z 296.88,A -85,B 0,C 180,E1 -16853.571,E2 -16853.571} C_VEL
LIN {X 0,Y 303.435,Z 284.498,A -85,B 0,C 180,E1 -16854.093,E2 -16854.093} C_VEL
LIN {X 0,Y 305.364,Z 212.457,A -85,B 0,C 180,E1 -16855.8,E2 -16855.8} C_VEL
LIN {X 0,Y 303.413,Z 201.897,A -85,B 0,C 180,E1 -16856.252,E2 -16856.252} C_VEL
LIN {X 0,Y 295.785,Z 182.979,A -85,B 0,C 180,E1 -16857.495,E2 -16857.495} C_VEL
LIN {X 0,Y 293.098,Z 176.891,A -85,B 0,C 180,E1 -16857.947,E2 -16857.947} C_VEL
LIN {X 0,Y 291.367,Z 169.693,A -85,B 0,C 180,E1 -16860.634,E2 -16860.634} C_VEL
LIN {X 0,Y 291.371,Z 169.687,A -85,B 0,C 180,E1 -16864.905,E2 -16864.905} C_VEL
LIN {X 0,Y 291.377,Z 169.687,A -85,B 0,C 180,E1 -16867.254,E2 -16867.254} C_VEL
LIN {X 0,Y 291.333,Z 169.696,A -85,B 0,C 180,E1 -16870.642,E2 -16870.642} C_VEL
LIN {X 0,Y 291.291,Z 169.699,A -85,B 0,C 180,E1 -16874.402,E2 -16874.402} C_VEL
LIN {X 0,Y 291.326,Z 169.694,A -85,B 0,C 180,E1 -16878.404,E2 -16878.404} C_VEL
LIN {X 0,Y 291.364,Z 169.688,A -85,B 0,C 180,E1 -16881.16,E2 -16881.16} C_VEL
LIN {X 0,Y 291.362,Z 169.689,A -85,B 0,C 180,E1 -16884.626,E2 -16884.626} C_VEL
LIN {X 0,Y 291.331,Z 169.688,A -85,B 0,C 180,E1 -16886.607,E2 -16886.607} C_VEL
LIN {X 0,Y 290.636,Z 169.779,A -85,B 0,C 180,E1 -16887.762,E2 -16887.762} C_VEL
LIN {X 0,Y 287.76,Z 170.142,A -85,B 0,C 180,E1 -16889.643,E2 -16889.643} C_VEL
LIN {X 0,Y 285.382,Z 170.433,A -85,B 0,C 180,E1 -16891.17,E2 -16891.17} C_VEL
LIN {X 0,Y 284.431,Z 170.549,A -85,B 0,C 180,E1 -16892.353,E2 -16892.353} C_VEL
LIN {X 0,Y 284.389,Z 170.554,A -85,B 0,C 180,E1 -16892.753,E2 -16892.753} C_VEL
LIN {X 0,Y 284.366,Z 170.559,A -85,B 0,C 180,E1 -16896.707,E2 -16896.707} C_VEL
LIN {X 0,Y 284.404,Z 170.56,A -85,B 0,C 180,E1 -16901.261,E2 -16901.261} C_VEL
LIN {X 0,Y 284.492,Z 170.537,A -85,B 0,C 180,E1 -16904.459,E2 -16904.459} C_VEL
LIN {X 0,Y 284.488,Z 170.547,A -85,B 0,C 180,E1 -16908.601,E2 -16908.601} C_VEL
LIN {X 0,Y 284.656,Z 170.519,A -85,B 0,C 180,E1 -16911.481,E2 -16911.481} C_VEL
LIN {X 0,Y 284.598,Z 170.532,A -85,B 0,C 180,E1 -16914.331,E2 -16914.331} C_VEL
LIN {X 0,Y 284.854,Z 170.495,A -85,B 0,C 180,E1 -16918.586,E2 -16918.586} C_VEL
LIN {X 0,Y 284.855,Z 170.501,A -85,B 0,C 180,E1 -16921.414,E2 -16921.414} C_VEL
LIN {X 0,Y 284.693,Z 170.518,A -85,B 0,C 180,E1 -16927.09,E2 -16927.09} C_VEL
LIN {X 0,Y 284.566,Z 170.537,A -85,B 0,C 180,E1 -16929.955,E2 -16929.955} C_VEL
LIN {X 0,Y 284.481,Z 170.543,A -85,B 0,C 180,E1 -16934.303,E2 -16934.303} C_VEL
LIN {X 0,Y 284.422,Z 170.553,A -85,B 0,C 180,E1 -16937.249,E2 -16937.249} C_VEL
LIN {X 0,Y 284.377,Z 170.557,A -85,B 0,C 180,E1 -16940.242,E2 -16940.242} C_VEL
LIN {X 0,Y 284.337,Z 170.559,A -85,B 0,C 180,E1 -16944.847,E2 -16944.847} C_VEL
LIN {X 0,Y 284.328,Z 170.569,A -85,B 0,C 180,E1 -16948.011,E2 -16948.011} C_VEL
LIN {X 0,Y 284.294,Z 170.569,A -85,B 0,C 180,E1 -16951.275,E2 -16951.275} C_VEL
LIN {X 0,Y 284.34,Z 170.563,A -85,B 0,C 180,E1 -16955.348,E2 -16955.348} C_VEL
LIN {X 0,Y 284.308,Z 170.567,A -85,B 0,C 180,E1 -16958.17,E2 -16958.17} C_VEL
LIN {X 0,Y 284.269,Z 170.575,A -85,B 0,C 180,E1 -16962.125,E2 -16962.125} C_VEL
LIN {X 0,Y 284.255,Z 170.575,A -85,B 0,C 180,E1 -16966.189,E2 -16966.189} C_VEL
LIN {X 0,Y 284.283,Z 170.572,A -85,B 0,C 180,E1 -16970.03,E2 -16970.03} C_VEL
LIN {X 0,Y 284.329,Z 170.567,A -85,B 0,C 180,E1 -16973.614,E2 -16973.614} C_VEL
LIN {X 0,Y 284.333,Z 170.615,A -85,B 0,C 180,E1 -16975.267,E2 -16975.267} C_VEL
LIN {X 0,Y 286.771,Z 181.076,A -85,B 0,C 180,E1 -16979.066,E2 -16979.066} C_VEL
LIN {X 0,Y 288.28,Z 188.505,A -85,B 0,C 180,E1 -16981.599,E2 -16981.599} C_VEL
LIN {X 0,Y 293.26,Z 201.148,A -85,B 0,C 180,E1 -16982.463,E2 -16982.463} C_VEL
LIN {X 0,Y 297.508,Z 225.837,A -85,B 0,C 180,E1 -16983.539,E2 -16983.539} C_VEL
LIN {X 0,Y 298.444,Z 233.049,A -85,B 0,C 180,E1 -16983.817,E2 -16983.817} C_VEL
LIN {X 0,Y 296.638,Z 297.009,A -85,B 0,C 180,E1 -16985.365,E2 -16985.365} C_VEL
LIN {X 0,Y 295.664,Z 310.16,A -85,B 0,C 180,E1 -16985.933,E2 -16985.933} C_VEL
LIN {X 0,Y 294.497,Z 322.258,A -85,B 0,C 180,E1 -16986.718,E2 -16986.718} C_VEL
LIN {X 0,Y 292.946,Z 334.471,A -85,B 0,C 180,E1 -16987.799,E2 -16987.799} C_VEL
LIN {X 0,Y 291.119,Z 346.036,A -85,B 0,C 180,E1 -16989.14,E2 -16989.14} C_VEL
LIN {X 0,Y 289.332,Z 356.453,A -85,B 0,C 180,E1 -16990.673,E2 -16990.673} C_VEL
LIN {X 0,Y 287.713,Z 366.193,A -85,B 0,C 180,E1 -16992.487,E2 -16992.487} C_VEL
LIN {X 0,Y 286.212,Z 374.209,A -85,B 0,C 180,E1 -16994.329,E2 -16994.329} C_VEL
LIN {X 0,Y 284.759,Z 381.63,A -85,B 0,C 180,E1 -16996.44,E2 -16996.44} C_VEL
LIN {X 0,Y 283.728,Z 387.594,A -85,B 0,C 180,E1 -16998.571,E2 -16998.571} C_VEL
LIN {X 0,Y 282.99,Z 392.307,A -85,B 0,C 180,E1 -17000.71,E2 -17000.71} C_VEL
LIN {X 0,Y 282.554,Z 395.909,A -85,B 0,C 180,E1 -17002.856,E2 -17002.856} C_VEL
LIN {X 0,Y 282.336,Z 398.176,A -85,B 0,C 180,E1 -17004.683,E2 -17004.683} C_VEL
LIN {X 0,Y 282.332,Z 400.157,A -85,B 0,C 180,E1 -17007.146,E2 -17007.146} C_VEL
LIN {X 0,Y 282.322,Z 400.763,A -85,B 0,C 180,E1 -17008.574,E2 -17008.574} C_VEL
LIN {X 0,Y 282.322,Z 400.976,A -85,B 0,C 180,E1 -17010,E2 -17010} C_VEL
LIN {X 0,Y 282.322,Z 400.755,A -85,B 0,C 180,E1 -17011.426,E2 -17011.426} C_VEL
LIN {X 0,Y 282.332,Z 400.143,A -85,B 0,C 180,E1 -17012.854,E2 -17012.854} C_VEL
LIN {X 0,Y 282.386,Z 397.739,A -85,B 0,C 180,E1 -17015.713,E2 -17015.713} C_VEL
LIN {X 0,Y 282.676,Z 394.797,A -85,B 0,C 180,E1 -17017.859,E2 -17017.859} C_VEL
LIN {X 0,Y 283.21,Z 390.817,A -85,B 0,C 180,E1 -17020.004,E2 -17020.004} C_VEL
LIN {X 0,Y 284.155,Z 384.698,A -85,B 0,C 180,E1 -17022.498,E2 -17022.498} C_VEL
LIN {X 0,Y 285.456,Z 378.021,A -85,B 0,C 180,E1 -17024.617,E2 -17024.617} C_VEL
LIN {X 0,Y 287,Z 369.736,A -85,B 0,C 180,E1 -17026.722,E2 -17026.722} C_VEL
LIN {X 0,Y 288.451,Z 361.238,A -85,B 0,C 180,E1 -17028.466,E2 -17028.466} C_VEL
LIN {X 0,Y 290.269,Z 350.742,A -85,B 0,C 180,E1 -17030.183,E2 -17030.183} C_VEL
LIN {X 0,Y 291.979,Z 340.359,A -85,B 0,C 180,E1 -17031.535,E2 -17031.535} C_VEL
LIN {X 0,Y 293.588,Z 328.968,A -85,B 0,C 180,E1 -17032.706,E2 -17032.706} C_VEL
LIN {X 0,Y 294.955,Z 317.245,A -85,B 0,C 180,E1 -17033.616,E2 -17033.616} C_VEL
LIN {X 0,Y 296.139,Z 304.643,A -85,B 0,C 180,E1 -17034.306,E2 -17034.306} C_VEL
LIN {X 0,Y 296.902,Z 291.782,A -85,B 0,C 180,E1 -17034.751,E2 -17034.751} C_VEL
LIN {X 0,Y 298.298,Z 231.494,A -85,B 0,C 180,E1 -17036.206,E2 -17036.206} C_VEL
LIN {X 0,Y 294.205,Z 206.498,A -85,B 0,C 180,E1 -17037.265,E2 -17037.265} C_VEL
LIN {X 0,Y 292.671,Z 199.473,A -85,B 0,C 180,E1 -17037.609,E2 -17037.609} C_VEL
LIN {X 0,Y 288.27,Z 188.35,A -85,B 0,C 180,E1 -17038.395,E2 -17038.395} C_VEL
LIN {X 0,Y 286.174,Z 178.32,A -85,B 0,C 180,E1 -17041.871,E2 -17041.871} C_VEL
LIN {X 0,Y 284.332,Z 170.569,A -85,B 0,C 180,E1 -17044.733,E2 -17044.733} C_VEL
LIN {X 0,Y 284.301,Z 170.572,A -85,B 0,C 180,E1 -17048.171,E2 -17048.171} C_VEL
LIN {X 0,Y 284.237,Z 170.58,A -85,B 0,C 180,E1 -17052.117,E2 -17052.117} C_VEL
LIN {X 0,Y 284.256,Z 170.578,A -85,B 0,C 180,E1 -17056.189,E2 -17056.189} C_VEL
LIN {X 0,Y 284.306,Z 170.571,A -85,B 0,C 180,E1 -17060.024,E2 -17060.024} C_VEL
LIN {X 0,Y 284.33,Z 170.566,A -85,B 0,C 180,E1 -17063.614,E2 -17063.614} C_VEL
LIN {X 0,Y 284.306,Z 170.569,A -85,B 0,C 180,E1 -17067.19,E2 -17067.19} C_VEL
LIN {X 0,Y 284.34,Z 170.567,A -85,B 0,C 180,E1 -17070.374,E2 -17070.374} C_VEL
LIN {X 0,Y 284.314,Z 170.566,A -85,B 0,C 180,E1 -17073.58,E2 -17073.58} C_VEL
LIN {X 0,Y 284.331,Z 170.563,A -85,B 0,C 180,E1 -17076.704,E2 -17076.704} C_VEL
LIN {X 0,Y 284.399,Z 170.557,A -85,B 0,C 180,E1 -17081.261,E2 -17081.261} C_VEL
LIN {X 0,Y 284.492,Z 170.546,A -85,B 0,C 180,E1 -17084.459,E2 -17084.459} C_VEL
LIN {X 0,Y 284.487,Z 170.543,A -85,B 0,C 180,E1 -17088.601,E2 -17088.601} C_VEL
LIN {X 0,Y 284.639,Z 170.53,A -85,B 0,C 180,E1 -17091.481,E2 -17091.481} C_VEL
LIN {X 0,Y 284.597,Z 170.529,A -85,B 0,C 180,E1 -17094.331,E2 -17094.331} C_VEL
LIN {X 0,Y 284.856,Z 170.498,A -85,B 0,C 180,E1 -17098.586,E2 -17098.586} C_VEL
LIN {X 0,Y 284.855,Z 170.503,A -85,B 0,C 180,E1 -17101.414,E2 -17101.414} C_VEL
LIN {X 0,Y 284.686,Z 170.522,A -85,B 0,C 180,E1 -17107.09,E2 -17107.09} C_VEL
LIN {X 0,Y 284.519,Z 170.541,A -85,B 0,C 180,E1 -17109.957,E2 -17109.957} C_VEL
LIN {X 0,Y 284.482,Z 170.548,A -85,B 0,C 180,E1 -17114.303,E2 -17114.303} C_VEL
LIN {X 0,Y 284.426,Z 170.55,A -85,B 0,C 180,E1 -17117.248,E2 -17117.248} C_VEL
LIN {X 0,Y 284.379,Z 170.561,A -85,B 0,C 180,E1 -17120.242,E2 -17120.242} C_VEL
LIN {X 0,Y 284.37,Z 170.559,A -85,B 0,C 180,E1 -17123.876,E2 -17123.876} C_VEL
LIN {X 0,Y 284.398,Z 170.553,A -85,B 0,C 180,E1 -17127.174,E2 -17127.174} C_VEL
LIN {X 0,Y 284.296,Z 170.568,A -85,B 0,C 180,E1 -17131.274,E2 -17131.274} C_VEL
LIN {X 0,Y 284.362,Z 170.561,A -85,B 0,C 180,E1 -17135.354,E2 -17135.354} C_VEL
LIN {X 0,Y 284.323,Z 170.569,A -85,B 0,C 180,E1 -17138.167,E2 -17138.167} C_VEL
LIN {X 0,Y 284.27,Z 170.574,A -85,B 0,C 180,E1 -17142.125,E2 -17142.125} C_VEL
LIN {X 0,Y 284.256,Z 170.577,A -85,B 0,C 180,E1 -17146.19,E2 -17146.19} C_VEL
LIN {X 0,Y 284.308,Z 170.57,A -85,B 0,C 180,E1 -17150.024,E2 -17150.024} C_VEL
LIN {X 0,Y 284.336,Z 170.57,A -85,B 0,C 180,E1 -17153.615,E2 -17153.615} C_VEL
LIN {X 0,Y 284.309,Z 170.568,A -85,B 0,C 180,E1 -17157.19,E2 -17157.19} C_VEL
LIN {X 0,Y 284.334,Z 170.589,A -85,B 0,C 180,E1 -17158.959,E2 -17158.959} C_VEL
LIN {X 0,Y 285.905,Z 177.142,A -85,B 0,C 180,E1 -17161.427,E2 -17161.427} C_VEL
LIN {X 0,Y 293.258,Z 194.005,A -85,B 0,C 180,E1 -17162.669,E2 -17162.669} C_VEL
LIN {X 0,Y 297.611,Z 205.661,A -85,B 0,C 180,E1 -17163.414,E2 -17163.414} C_VEL
LIN {X 0,Y 298.908,Z 212.608,A -85,B 0,C 180,E1 -17163.722,E2 -17163.722} C_VEL
LIN {X 0,Y 297.03,Z 282.512,A -85,B 0,C 180,E1 -17165.4,E2 -17165.4} C_VEL
LIN {X 0,Y 296.283,Z 295.029,A -85,B 0,C 180,E1 -17165.893,E2 -17165.893} C_VEL
LIN {X 0,Y 295.182,Z 307.828,A -85,B 0,C 180,E1 -17166.683,E2 -17166.683} C_VEL
LIN {X 0,Y 293.808,Z 319.678,A -85,B 0,C 180,E1 -17167.683,E2 -17167.683} C_VEL
LIN {X 0,Y 292.327,Z 330.43,A -85,B 0,C 180,E1 -17168.862,E2 -17168.862} C_VEL
LIN {X 0,Y 290.742,Z 340.316,A -85,B 0,C 180,E1 -17170.22,E2 -17170.22} C_VEL
LIN {X 0,Y 289.241,Z 350.285,A -85,B 0,C 180,E1 -17171.953,E2 -17171.953} C_VEL
LIN {X 0,Y 287.342,Z 359.934,A -85,B 0,C 180,E1 -17174.028,E2 -17174.028} C_VEL
LIN {X 0,Y 285.804,Z 367.627,A -85,B 0,C 180,E1 -17176.128,E2 -17176.128} C_VEL
LIN {X 0,Y 284.437,Z 374.687,A -85,B 0,C 180,E1 -17178.599,E2 -17178.599} C_VEL
LIN {X 0,Y 283.546,Z 379.389,A -85,B 0,C 180,E1 -17180.729,E2 -17180.729} C_VEL
LIN {X 0,Y 283.052,Z 382.984,A -85,B 0,C 180,E1 -17182.868,E2 -17182.868} C_VEL
LIN {X 0,Y 282.765,Z 384.842,A -85,B 0,C 180,E1 -17184.294,E2 -17184.294} C_VEL
LIN {X 0,Y 282.595,Z 386.239,A -85,B 0,C 180,E1 -17185.721,E2 -17185.721} C_VEL
LIN {X 0,Y 282.477,Z 387.232,A -85,B 0,C 180,E1 -17187.148,E2 -17187.148} C_VEL
LIN {X 0,Y 282.329,Z 388.076,A -85,B 0,C 180,E1 -17190,E2 -17190} C_VEL
LIN {X 0,Y 282.365,Z 387.884,A -85,B 0,C 180,E1 -17191.426,E2 -17191.426} C_VEL
LIN {X 0,Y 282.476,Z 387.296,A -85,B 0,C 180,E1 -17192.852,E2 -17192.852} C_VEL
LIN {X 0,Y 282.587,Z 386.328,A -85,B 0,C 180,E1 -17194.279,E2 -17194.279} C_VEL
LIN {X 0,Y 282.817,Z 384.28,A -85,B 0,C 180,E1 -17196.276,E2 -17196.276} C_VEL
LIN {X 0,Y 283.356,Z 380.904,A -85,B 0,C 180,E1 -17198.558,E2 -17198.558} C_VEL
LIN {X 0,Y 284.08,Z 376.648,A -85,B 0,C 180,E1 -17200.693,E2 -17200.693} C_VEL
LIN {X 0,Y 285.369,Z 370.201,A -85,B 0,C 180,E1 -17203.168,E2 -17203.168} C_VEL
LIN {X 0,Y 286.692,Z 363.117,A -85,B 0,C 180,E1 -17205.279,E2 -17205.279} C_VEL
LIN {X 0,Y 288.528,Z 354.286,A -85,B 0,C 180,E1 -17207.361,E2 -17207.361} C_VEL
LIN {X 0,Y 290.113,Z 344.697,A -85,B 0,C 180,E1 -17209.188,E2 -17209.188} C_VEL
LIN {X 0,Y 291.845,Z 333.905,A -85,B 0,C 180,E1 -17210.805,E2 -17210.805} C_VEL
LIN {X 0,Y 293.525,Z 322.449,A -85,B 0,C 180,E1 -17212.155,E2 -17212.155} C_VEL
LIN {X 0,Y 295.037,Z 310.433,A -85,B 0,C 180,E1 -17213.237,E2 -17213.237} C_VEL
LIN {X 0,Y 296.131,Z 297.032,A -85,B 0,C 180,E1 -17214.12,E2 -17214.12} C_VEL
LIN {X 0,Y 296.988,Z 284.645,A -85,B 0,C 180,E1 -17214.65,E2 -17214.65} C_VEL
LIN {X 0,Y 298.893,Z 212.329,A -85,B 0,C 180,E1 -17216.408,E2 -17216.408} C_VEL
LIN {X 0,Y 297.157,Z 203.972,A -85,B 0,C 180,E1 -17216.797,E2 -17216.797} C_VEL
LIN {X 0,Y 289.688,Z 185.547,A -85,B 0,C 180,E1 -17218.057,E2 -17218.057} C_VEL
LIN {X 0,Y 285.843,Z 177.018,A -85,B 0,C 180,E1 -17218.74,E2 -17218.74} C_VEL
LIN {X 0,Y 284.341,Z 170.568,A -85,B 0,C 180,E1 -17221.194,E2 -17221.194} C_VEL
LIN {X 0,Y 284.342,Z 170.564,A -85,B 0,C 180,E1 -17225.348,E2 -17225.348} C_VEL
LIN {X 0,Y 284.313,Z 170.57,A -85,B 0,C 180,E1 -17228.169,E2 -17228.169} C_VEL
LIN {X 0,Y 284.27,Z 170.575,A -85,B 0,C 180,E1 -17232.124,E2 -17232.124} C_VEL
LIN {X 0,Y 284.256,Z 170.579,A -85,B 0,C 180,E1 -17236.189,E2 -17236.189} C_VEL
LIN {X 0,Y 284.307,Z 170.572,A -85,B 0,C 180,E1 -17240.023,E2 -17240.023} C_VEL
LIN {X 0,Y 284.336,Z 170.565,A -85,B 0,C 180,E1 -17243.614,E2 -17243.614} C_VEL
LIN {X 0,Y 284.308,Z 170.563,A -85,B 0,C 180,E1 -17247.189,E2 -17247.189} C_VEL
LIN {X 0,Y 284.359,Z 170.56,A -85,B 0,C 180,E1 -17250.376,E2 -17250.376} C_VEL
LIN {X 0,Y 284.389,Z 170.554,A -85,B 0,C 180,E1 -17252.753,E2 -17252.753} C_VEL
LIN {X 0,Y 284.135,Z 170.59,A -85,B 0,C 180,E1 -17253.543,E2 -17253.543} C_VEL
LIN {X 0,Y 282.803,Z 170.757,A -85,B 0,C 180,E1 -17254.709,E2 -17254.709} C_VEL
LIN {X 0,Y 278.388,Z 171.302,A -85,B 0,C 180,E1 -17257.417,E2 -17257.417} C_VEL
LIN {X 0,Y 277.346,Z 171.43,A -85,B 0,C 180,E1 -17258.63,E2 -17258.63} C_VEL
LIN {X 0,Y 277.282,Z 171.439,A -85,B 0,C 180,E1 -17259.041,E2 -17259.041} C_VEL
LIN {X 0,Y 277.361,Z 171.433,A -85,B 0,C 180,E1 -17262.298,E2 -17262.298} C_VEL
LIN {X 0,Y 277.434,Z 171.42,A -85,B 0,C 180,E1 -17265.326,E2 -17265.326} C_VEL
LIN {X 0,Y 277.506,Z 171.412,A -85,B 0,C 180,E1 -17269.789,E2 -17269.789} C_VEL
LIN {X 0,Y 277.648,Z 171.393,A -85,B 0,C 180,E1 -17272.729,E2 -17272.729} C_VEL
LIN {X 0,Y 277.82,Z 171.37,A -85,B 0,C 180,E1 -17278.55,E2 -17278.55} C_VEL
LIN {X 0,Y 277.821,Z 171.377,A -85,B 0,C 180,E1 -17281.449,E2 -17281.449} C_VEL
LIN {X 0,Y 277.648,Z 171.395,A -85,B 0,C 180,E1 -17287.271,E2 -17287.271} C_VEL
LIN {X 0,Y 277.506,Z 171.418,A -85,B 0,C 180,E1 -17290.211,E2 -17290.211} C_VEL
LIN {X 0,Y 277.434,Z 171.424,A -85,B 0,C 180,E1 -17294.674,E2 -17294.674} C_VEL
LIN {X 0,Y 277.342,Z 171.429,A -85,B 0,C 180,E1 -17299.234,E2 -17299.234} C_VEL
LIN {X 0,Y 277.292,Z 171.44,A -85,B 0,C 180,E1 -17304.158,E2 -17304.158} C_VEL
LIN {X 0,Y 277.324,Z 171.439,A -85,B 0,C 180,E1 -17307.505,E2 -17307.505} C_VEL
LIN {X 0,Y 277.272,Z 171.443,A -85,B 0,C 180,E1 -17310.482,E2 -17310.482} C_VEL
LIN {X 0,Y 277.246,Z 171.447,A -85,B 0,C 180,E1 -17313.896,E2 -17313.896} C_VEL
LIN {X 0,Y 277.264,Z 171.448,A -85,B 0,C 180,E1 -17317.47,E2 -17317.47} C_VEL
LIN {X 0,Y 277.209,Z 171.454,A -85,B 0,C 180,E1 -17321.237,E2 -17321.237} C_VEL
LIN {X 0,Y 277.201,Z 171.455,A -85,B 0,C 180,E1 -17325.227,E2 -17325.227} C_VEL
LIN {X 0,Y 277.197,Z 171.456,A -85,B 0,C 180,E1 -17329.519,E2 -17329.519} C_VEL
LIN {X 0,Y 277.261,Z 171.448,A -85,B 0,C 180,E1 -17332.53,E2 -17332.53} C_VEL
LIN {X 0,Y 277.32,Z 171.625,A -85,B 0,C 180,E1 -17334.681,E2 -17334.681} C_VEL
LIN {X 0,Y 279.463,Z 180.764,A -85,B 0,C 180,E1 -17338.122,E2 -17338.122} C_VEL
LIN {X 0,Y 281.093,Z 188.454,A -85,B 0,C 180,E1 -17340.807,E2 -17340.807} C_VEL
LIN {X 0,Y 287.209,Z 203.717,A -85,B 0,C 180,E1 -17341.906,E2 -17341.906} C_VEL
LIN {X 0,Y 291.214,Z 227.088,A -85,B 0,C 180,E1 -17342.959,E2 -17342.959} C_VEL
LIN {X 0,Y 292.063,Z 233.716,A -85,B 0,C 180,E1 -17343.222,E2 -17343.222} C_VEL
LIN {X 0,Y 290.19,Z 296.86,A -85,B 0,C 180,E1 -17344.78,E2 -17344.78} C_VEL
LIN {X 0,Y 289.206,Z 310.007,A -85,B 0,C 180,E1 -17345.36,E2 -17345.36} C_VEL
LIN {X 0,Y 287.991,Z 322.102,A -85,B 0,C 180,E1 -17346.16,E2 -17346.16} C_VEL
LIN {X 0,Y 286.379,Z 334.313,A -85,B 0,C 180,E1 -17347.262,E2 -17347.262} C_VEL
LIN {X 0,Y 284.503,Z 345.878,A -85,B 0,C 180,E1 -17348.632,E2 -17348.632} C_VEL
LIN {X 0,Y 282.63,Z 356.293,A -85,B 0,C 180,E1 -17350.196,E2 -17350.196} C_VEL
LIN {X 0,Y 281.024,Z 365.191,A -85,B 0,C 180,E1 -17351.865,E2 -17351.865} C_VEL
LIN {X 0,Y 279.342,Z 374.047,A -85,B 0,C 180,E1 -17353.934,E2 -17353.934} C_VEL
LIN {X 0,Y 277.847,Z 381.469,A -85,B 0,C 180,E1 -17356.096,E2 -17356.096} C_VEL
LIN {X 0,Y 276.743,Z 387.432,A -85,B 0,C 180,E1 -17358.278,E2 -17358.278} C_VEL
LIN {X 0,Y 275.961,Z 392.145,A -85,B 0,C 180,E1 -17360.472,E2 -17360.472} C_VEL
LIN {X 0,Y 275.493,Z 395.747,A -85,B 0,C 180,E1 -17362.672,E2 -17362.672} C_VEL
LIN {X 0,Y 275.228,Z 398.262,A -85,B 0,C 180,E1 -17364.794,E2 -17364.794} C_VEL
LIN {X 0,Y 275.241,Z 399.995,A -85,B 0,C 180,E1 -17367.073,E2 -17367.073} C_VEL
LIN {X 0,Y 275.247,Z 400.602,A -85,B 0,C 180,E1 -17368.537,E2 -17368.537} C_VEL
LIN {X 0,Y 275.246,Z 400.814,A -85,B 0,C 180,E1 -17370,E2 -17370} C_VEL
LIN {X 0,Y 275.247,Z 400.593,A -85,B 0,C 180,E1 -17371.463,E2 -17371.463} C_VEL
LIN {X 0,Y 275.241,Z 399.981,A -85,B 0,C 180,E1 -17372.927,E2 -17372.927} C_VEL
LIN {X 0,Y 275.237,Z 398.216,A -85,B 0,C 180,E1 -17375.226,E2 -17375.226} C_VEL
LIN {X 0,Y 275.606,Z 394.633,A -85,B 0,C 180,E1 -17378.062,E2 -17378.062} C_VEL
LIN {X 0,Y 276.194,Z 390.653,A -85,B 0,C 180,E1 -17380.26,E2 -17380.26} C_VEL
LIN {X 0,Y 277.205,Z 384.534,A -85,B 0,C 180,E1 -17382.817,E2 -17382.817} C_VEL
LIN {X 0,Y 278.578,Z 377.857,A -85,B 0,C 180,E1 -17384.986,E2 -17384.986} C_VEL
LIN {X 0,Y 280.195,Z 369.572,A -85,B 0,C 180,E1 -17387.141,E2 -17387.141} C_VEL
LIN {X 0,Y 281.7,Z 361.073,A -85,B 0,C 180,E1 -17388.925,E2 -17388.925} C_VEL
LIN {X 0,Y 283.606,Z 350.576,A -85,B 0,C 180,E1 -17390.679,E2 -17390.679} C_VEL
LIN {X 0,Y 285.608,Z 338.762,A -85,B 0,C 180,E1 -17392.231,E2 -17392.231} C_VEL
LIN {X 0,Y 287.231,Z 326.859,A -85,B 0,C 180,E1 -17393.429,E2 -17393.429} C_VEL
LIN {X 0,Y 288.734,Z 314.472,A -85,B 0,C 180,E1 -17394.348,E2 -17394.348} C_VEL
LIN {X 0,Y 289.926,Z 301.713,A -85,B 0,C 180,E1 -17395.005,E2 -17395.005} C_VEL
LIN {X 0,Y 290.533,Z 288.211,A -85,B 0,C 180,E1 -17395.428,E2 -17395.428} C_VEL
LIN {X 0,Y 291.853,Z 231.972,A -85,B 0,C 180,E1 -17396.812,E2 -17396.812} C_VEL
LIN {X 0,Y 287.961,Z 207.929,A -85,B 0,C 180,E1 -17397.863,E2 -17397.863} C_VEL
LIN {X 0,Y 286.689,Z 202.149,A -85,B 0,C 180,E1 -17398.157,E2 -17398.157} C_VEL
LIN {X 0,Y 280.969,Z 188.145,A -85,B 0,C 180,E1 -17399.208,E2 -17399.208} C_VEL
LIN {X 0,Y 279.167,Z 179.387,A -85,B 0,C 180,E1 -17402.342,E2 -17402.342} C_VEL
LIN {X 0,Y 277.299,Z 171.444,A -85,B 0,C 180,E1 -17405.378,E2 -17405.378} C_VEL
LIN {X 0,Y 277.217,Z 171.454,A -85,B 0,C 180,E1 -17409.331,E2 -17409.331} C_VEL
LIN {X 0,Y 277.201,Z 171.456,A -85,B 0,C 180,E1 -17413.2,E2 -17413.2} C_VEL
LIN {X 0,Y 277.215,Z 171.452,A -85,B 0,C 180,E1 -17417.325,E2 -17417.325} C_VEL
LIN {X 0,Y 277.261,Z 171.448,A -85,B 0,C 180,E1 -17421.793,E2 -17421.793} C_VEL
LIN {X 0,Y 277.284,Z 171.447,A -85,B 0,C 180,E1 -17424.341,E2 -17424.341} C_VEL
LIN {X 0,Y 277.24,Z 171.451,A -85,B 0,C 180,E1 -17427.836,E2 -17427.836} C_VEL
LIN {X 0,Y 277.243,Z 171.449,A -85,B 0,C 180,E1 -17431.207,E2 -17431.207} C_VEL
LIN {X 0,Y 277.272,Z 171.446,A -85,B 0,C 180,E1 -17434.475,E2 -17434.475} C_VEL
LIN {X 0,Y 277.267,Z 171.444,A -85,B 0,C 180,E1 -17437.653,E2 -17437.653} C_VEL
LIN {X 0,Y 277.342,Z 171.435,A -85,B 0,C 180,E1 -17440.766,E2 -17440.766} C_VEL
LIN {X 0,Y 277.435,Z 171.427,A -85,B 0,C 180,E1 -17445.326,E2 -17445.326} C_VEL
LIN {X 0,Y 277.461,Z 171.424,A -85,B 0,C 180,E1 -17449.787,E2 -17449.787} C_VEL
LIN {X 0,Y 277.641,Z 171.397,A -85,B 0,C 180,E1 -17452.729,E2 -17452.729} C_VEL
LIN {X 0,Y 277.822,Z 171.374,A -85,B 0,C 180,E1 -17458.551,E2 -17458.551} C_VEL
LIN {X 0,Y 277.821,Z 171.379,A -85,B 0,C 180,E1 -17461.45,E2 -17461.45} C_VEL
LIN {X 0,Y 277.641,Z 171.401,A -85,B 0,C 180,E1 -17467.271,E2 -17467.271} C_VEL
LIN {X 0,Y 277.461,Z 171.42,A -85,B 0,C 180,E1 -17470.213,E2 -17470.213} C_VEL
LIN {X 0,Y 277.435,Z 171.428,A -85,B 0,C 180,E1 -17474.674,E2 -17474.674} C_VEL
LIN {X 0,Y 277.346,Z 171.437,A -85,B 0,C 180,E1 -17479.234,E2 -17479.234} C_VEL
LIN {X 0,Y 277.32,Z 171.439,A -85,B 0,C 180,E1 -17484.171,E2 -17484.171} C_VEL
LIN {X 0,Y 277.326,Z 171.434,A -85,B 0,C 180,E1 -17487.505,E2 -17487.505} C_VEL
LIN {X 0,Y 277.272,Z 171.446,A -85,B 0,C 180,E1 -17490.482,E2 -17490.482} C_VEL
LIN {X 0,Y 277.255,Z 171.449,A -85,B 0,C 180,E1 -17493.895,E2 -17493.895} C_VEL
LIN {X 0,Y 277.281,Z 171.444,A -85,B 0,C 180,E1 -17497.467,E2 -17497.467} C_VEL
LIN {X 0,Y 277.21,Z 171.453,A -85,B 0,C 180,E1 -17501.237,E2 -17501.237} C_VEL
LIN {X 0,Y 277.202,Z 171.453,A -85,B 0,C 180,E1 -17505.227,E2 -17505.227} C_VEL
LIN {X 0,Y 277.224,Z 171.454,A -85,B 0,C 180,E1 -17509.512,E2 -17509.512} C_VEL
LIN {X 0,Y 277.273,Z 171.447,A -85,B 0,C 180,E1 -17512.532,E2 -17512.532} C_VEL
LIN {X 0,Y 277.249,Z 171.448,A -85,B 0,C 180,E1 -17516.105,E2 -17516.105} C_VEL
LIN {X 0,Y 277.278,Z 171.569,A -85,B 0,C 180,E1 -17518.37,E2 -17518.37} C_VEL
LIN {X 0,Y 278.699,Z 177.308,A -85,B 0,C 180,E1 -17520.615,E2 -17520.615} C_VEL
LIN {X 0,Y 287.24,Z 196.625,A -85,B 0,C 180,E1 -17522.115,E2 -17522.115} C_VEL
LIN {X 0,Y 291.515,Z 207.991,A -85,B 0,C 180,E1 -17522.871,E2 -17522.871} C_VEL
LIN {X 0,Y 292.562,Z 213.877,A -85,B 0,C 180,E1 -17523.136,E2 -17523.136} C_VEL
LIN {X 0,Y 290.598,Z 282.695,A -85,B 0,C 180,E1 -17524.818,E2 -17524.818} C_VEL
LIN {X 0,Y 289.827,Z 295.202,A -85,B 0,C 180,E1 -17525.321,E2 -17525.321} C_VEL
LIN {X 0,Y 288.67,Z 307.998,A -85,B 0,C 180,E1 -17526.124,E2 -17526.124} C_VEL
LIN {X 0,Y 287.261,Z 319.846,A -85,B 0,C 180,E1 -17527.146,E2 -17527.146} C_VEL
LIN {X 0,Y 285.724,Z 330.597,A -85,B 0,C 180,E1 -17528.349,E2 -17528.349} C_VEL
LIN {X 0,Y 284.077,Z 340.482,A -85,B 0,C 180,E1 -17529.735,E2 -17529.735} C_VEL
LIN {X 0,Y 282.491,Z 350.451,A -85,B 0,C 180,E1 -17531.506,E2 -17531.506} C_VEL
LIN {X 0,Y 280.53,Z 360.099,A -85,B 0,C 180,E1 -17533.63,E2 -17533.63} C_VEL
LIN {X 0,Y 278.905,Z 367.791,A -85,B 0,C 180,E1 -17535.778,E2 -17535.778} C_VEL
LIN {X 0,Y 277.471,Z 374.851,A -85,B 0,C 180,E1 -17538.309,E2 -17538.309} C_VEL
LIN {X 0,Y 276.532,Z 379.553,A -85,B 0,C 180,E1 -17540.491,E2 -17540.491} C_VEL
LIN {X 0,Y 276.007,Z 383.147,A -85,B 0,C 180,E1 -17542.685,E2 -17542.685} C_VEL
LIN {X 0,Y 275.708,Z 385.005,A -85,B 0,C 180,E1 -17544.148,E2 -17544.148} C_VEL
LIN {X 0,Y 275.523,Z 386.401,A -85,B 0,C 180,E1 -17545.611,E2 -17545.611} C_VEL
LIN {X 0,Y 275.411,Z 387.394,A -85,B 0,C 180,E1 -17547.075,E2 -17547.075} C_VEL
LIN {X 0,Y 275.253,Z 388.238,A -85,B 0,C 180,E1 -17550,E2 -17550} C_VEL
LIN {X 0,Y 275.291,Z 388.045,A -85,B 0,C 180,E1 -17551.463,E2 -17551.463} C_VEL
LIN {X 0,Y 275.409,Z 387.458,A -85,B 0,C 180,E1 -17552.925,E2 -17552.925} C_VEL
LIN {X 0,Y 275.514,Z 386.49,A -85,B 0,C 180,E1 -17554.389,E2 -17554.389} C_VEL
LIN {X 0,Y 275.736,Z 384.66,A -85,B 0,C 180,E1 -17556.256,E2 -17556.256} C_VEL
LIN {X 0,Y 276.311,Z 381.066,A -85,B 0,C 180,E1 -17558.778,E2 -17558.778} C_VEL
LIN {X 0,Y 277.096,Z 376.809,A -85,B 0,C 180,E1 -17560.966,E2 -17560.966} C_VEL
LIN {X 0,Y 278.466,Z 370.361,A -85,B 0,C 180,E1 -17563.5,E2 -17563.5} C_VEL
LIN {X 0,Y 279.851,Z 363.277,A -85,B 0,C 180,E1 -17565.662,E2 -17565.662} C_VEL
LIN {X 0,Y 281.765,Z 354.445,A -85,B 0,C 180,E1 -17567.791,E2 -17567.791} C_VEL
LIN {X 0,Y 283.354,Z 345.183,A -85,B 0,C 180,E1 -17569.602,E2 -17569.602} C_VEL
LIN {X 0,Y 285.026,Z 335.351,A -85,B 0,C 180,E1 -17571.138,E2 -17571.138} C_VEL
LIN {X 0,Y 286.747,Z 324.184,A -85,B 0,C 180,E1 -17572.517,E2 -17572.517} C_VEL
LIN {X 0,Y 288.151,Z 313.63,A -85,B 0,C 180,E1 -17573.54,E2 -17573.54} C_VEL
LIN {X 0,Y 289.409,Z 300.914,A -85,B 0,C 180,E1 -17574.478,E2 -17574.478} C_VEL
LIN {X 0,Y 290.347,Z 288.21,A -85,B 0,C 180,E1 -17575.11,E2 -17575.11} C_VEL
LIN {X 0,Y 291.051,Z 271.98,A -85,B 0,C 180,E1 -17575.571,E2 -17575.571} C_VEL
LIN {X 0,Y 292.517,Z 213.345,A -85,B 0,C 180,E1 -17577.006,E2 -17577.006} C_VEL
LIN {X 0,Y 291.163,Z 206.657,A -85,B 0,C 180,E1 -17577.325,E2 -17577.325} C_VEL
LIN {X 0,Y 283.401,Z 187.456,A -85,B 0,C 180,E1 -17578.686,E2 -17578.686} C_VEL
LIN {X 0,Y 278.675,Z 177.25,A -85,B 0,C 180,E1 -17579.533,E2 -17579.533} C_VEL
LIN {X 0,Y 277.258,Z 171.45,A -85,B 0,C 180,E1 -17581.851,E2 -17581.851} C_VEL
LIN {X 0,Y 277.282,Z 171.444,A -85,B 0,C 180,E1 -17585.799,E2 -17585.799} C_VEL
LIN {X 0,Y 277.235,Z 171.449,A -85,B 0,C 180,E1 -17589.328,E2 -17589.328} C_VEL
LIN {X 0,Y 277.21,Z 171.454,A -85,B 0,C 180,E1 -17593.198,E2 -17593.198} C_VEL
LIN {X 0,Y 277.215,Z 171.452,A -85,B 0,C 180,E1 -17597.325,E2 -17597.325} C_VEL
LIN {X 0,Y 277.272,Z 171.443,A -85,B 0,C 180,E1 -17601.79,E2 -17601.79} C_VEL
LIN {X 0,Y 277.286,Z 171.444,A -85,B 0,C 180,E1 -17604.341,E2 -17604.341} C_VEL
LIN {X 0,Y 277.245,Z 171.447,A -85,B 0,C 180,E1 -17607.836,E2 -17607.836} C_VEL
LIN {X 0,Y 277.289,Z 171.441,A -85,B 0,C 180,E1 -17611.212,E2 -17611.212} C_VEL
LIN {X 0,Y 277.314,Z 171.44,A -85,B 0,C 180,E1 -17614.479,E2 -17614.479} C_VEL
LIN {X 0,Y 277.285,Z 171.438,A -85,B 0,C 180,E1 -17617.655,E2 -17617.655} C_VEL
LIN {X 0,Y 277.282,Z 171.439,A -85,B 0,C 180,E1 -17619.041,E2 -17619.041} C_VEL
LIN {X 0,Y 276.686,Z 171.52,A -85,B 0,C 180,E1 -17620.254,E2 -17620.254} C_VEL
LIN {X 0,Y 273.917,Z 171.862,A -85,B 0,C 180,E1 -17622.232,E2 -17622.232} C_VEL
LIN {X 0,Y 271.517,Z 172.155,A -85,B 0,C 180,E1 -17623.84,E2 -17623.84} C_VEL
LIN {X 0,Y 270.461,Z 172.286,A -85,B 0,C 180,E1 -17625.084,E2 -17625.084} C_VEL
LIN {X 0,Y 270.364,Z 172.297,A -85,B 0,C 180,E1 -17625.506,E2 -17625.506} C_VEL
LIN {X 0,Y 270.441,Z 172.293,A -85,B 0,C 180,E1 -17629.519,E2 -17629.519} C_VEL
LIN {X 0,Y 270.607,Z 172.268,A -85,B 0,C 180,E1 -17632.539,E2 -17632.539} C_VEL
LIN {X 0,Y 270.786,Z 172.246,A -85,B 0,C 180,E1 -17638.513,E2 -17638.513} C_VEL
LIN {X 0,Y 270.787,Z 172.253,A -85,B 0,C 180,E1 -17641.487,E2 -17641.487} C_VEL
LIN {X 0,Y 270.607,Z 172.271,A -85,B 0,C 180,E1 -17647.461,E2 -17647.461} C_VEL
LIN {X 0,Y 270.441,Z 172.298,A -85,B 0,C 180,E1 -17650.481,E2 -17650.481} C_VEL
LIN {X 0,Y 270.402,Z 172.299,A -85,B 0,C 180,E1 -17655.065,E2 -17655.065} C_VEL
LIN {X 0,Y 270.299,Z 172.306,A -85,B 0,C 180,E1 -17659.756,E2 -17659.756} C_VEL
LIN {X 0,Y 270.237,Z 172.315,A -85,B 0,C 180,E1 -17664.589,E2 -17664.589} C_VEL
LIN {X 0,Y 270.269,Z 172.321,A -85,B 0,C 180,E1 -17667.909,E2 -17667.909} C_VEL
LIN {X 0,Y 270.184,Z 172.326,A -85,B 0,C 180,E1 -17671.348,E2 -17671.348} C_VEL
LIN {X 0,Y 270.201,Z 172.322,A -85,B 0,C 180,E1 -17674.906,E2 -17674.906} C_VEL
LIN {X 0,Y 270.197,Z 172.324,A -85,B 0,C 180,E1 -17678.711,E2 -17678.711} C_VEL
LIN {X 0,Y 270.165,Z 172.334,A -85,B 0,C 180,E1 -17683.249,E2 -17683.249} C_VEL
LIN {X 0,Y 270.154,Z 172.334,A -85,B 0,C 180,E1 -17687.439,E2 -17687.439} C_VEL
LIN {X 0,Y 270.207,Z 172.327,A -85,B 0,C 180,E1 -17691.374,E2 -17691.374} C_VEL
LIN {X 0,Y 270.237,Z 172.347,A -85,B 0,C 180,E1 -17693.945,E2 -17693.945} C_VEL
LIN {X 0,Y 272.197,Z 180.575,A -85,B 0,C 180,E1 -17697.166,E2 -17697.166} C_VEL
LIN {X 0,Y 273.884,Z 188.292,A -85,B 0,C 180,E1 -17699.961,E2 -17699.961} C_VEL
LIN {X 0,Y 281.186,Z 206.195,A -85,B 0,C 180,E1 -17701.324,E2 -17701.324} C_VEL
LIN {X 0,Y 284.99,Z 228.814,A -85,B 0,C 180,E1 -17702.37,E2 -17702.37} C_VEL
LIN {X 0,Y 285.687,Z 234.799,A -85,B 0,C 180,E1 -17702.609,E2 -17702.609} C_VEL
LIN {X 0,Y 283.796,Z 296.711,A -85,B 0,C 180,E1 -17704.171,E2 -17704.171} C_VEL
LIN {X 0,Y 282.754,Z 309.853,A -85,B 0,C 180,E1 -17704.759,E2 -17704.759} C_VEL
LIN {X 0,Y 281.516,Z 321.947,A -85,B 0,C 180,E1 -17705.577,E2 -17705.577} C_VEL
LIN {X 0,Y 279.842,Z 334.156,A -85,B 0,C 180,E1 -17706.7,E2 -17706.7} C_VEL
LIN {X 0,Y 277.91,Z 345.72,A -85,B 0,C 180,E1 -17708.099,E2 -17708.099} C_VEL
LIN {X 0,Y 275.949,Z 356.134,A -85,B 0,C 180,E1 -17709.696,E2 -17709.696} C_VEL
LIN {X 0,Y 274.15,Z 365.641,A -85,B 0,C 180,E1 -17711.536,E2 -17711.536} C_VEL
LIN {X 0,Y 272.483,Z 373.886,A -85,B 0,C 180,E1 -17713.518,E2 -17713.518} C_VEL
LIN {X 0,Y 270.949,Z 381.309,A -85,B 0,C 180,E1 -17715.735,E2 -17715.735} C_VEL
LIN {X 0,Y 269.741,Z 387.27,A -85,B 0,C 180,E1 -17717.969,E2 -17717.969} C_VEL
LIN {X 0,Y 268.946,Z 391.984,A -85,B 0,C 180,E1 -17720.221,E2 -17720.221} C_VEL
LIN {X 0,Y 268.417,Z 395.585,A -85,B 0,C 180,E1 -17722.478,E2 -17722.478} C_VEL
LIN {X 0,Y 268.123,Z 398.344,A -85,B 0,C 180,E1 -17724.907,E2 -17724.907} C_VEL
LIN {X 0,Y 268.152,Z 399.833,A -85,B 0,C 180,E1 -17726.995,E2 -17726.995} C_VEL
LIN {X 0,Y 268.174,Z 400.44,A -85,B 0,C 180,E1 -17728.498,E2 -17728.498} C_VEL
LIN {X 0,Y 268.171,Z 400.652,A -85,B 0,C 180,E1 -17730,E2 -17730} C_VEL
LIN {X 0,Y 268.174,Z 400.431,A -85,B 0,C 180,E1 -17731.502,E2 -17731.502} C_VEL
LIN {X 0,Y 268.152,Z 399.818,A -85,B 0,C 180,E1 -17733.005,E2 -17733.005} C_VEL
LIN {X 0,Y 268.163,Z 398.225,A -85,B 0,C 180,E1 -17735.188,E2 -17735.188} C_VEL
LIN {X 0,Y 268.553,Z 394.469,A -85,B 0,C 180,E1 -17738.276,E2 -17738.276} C_VEL
LIN {X 0,Y 269.193,Z 390.49,A -85,B 0,C 180,E1 -17740.53,E2 -17740.53} C_VEL
LIN {X 0,Y 270.265,Z 384.37,A -85,B 0,C 180,E1 -17743.152,E2 -17743.152} C_VEL
LIN {X 0,Y 271.716,Z 377.693,A -85,B 0,C 180,E1 -17745.374,E2 -17745.374} C_VEL
LIN {X 0,Y 273.396,Z 369.407,A -85,B 0,C 180,E1 -17747.581,E2 -17747.581} C_VEL
LIN {X 0,Y 274.973,Z 360.907,A -85,B 0,C 180,E1 -17749.406,E2 -17749.406} C_VEL
LIN {X 0,Y 276.95,Z 350.41,A -85,B 0,C 180,E1 -17751.199,E2 -17751.199} C_VEL
LIN {X 0,Y 279.052,Z 338.596,A -85,B 0,C 180,E1 -17752.782,E2 -17752.782} C_VEL
LIN {X 0,Y 280.716,Z 326.691,A -85,B 0,C 180,E1 -17754.006,E2 -17754.006} C_VEL
LIN {X 0,Y 282.283,Z 314.303,A -85,B 0,C 180,E1 -17754.941,E2 -17754.941} C_VEL
LIN {X 0,Y 283.5,Z 301.539,A -85,B 0,C 180,E1 -17755.612,E2 -17755.612} C_VEL
LIN {X 0,Y 284.138,Z 288.027,A -85,B 0,C 180,E1 -17756.042,E2 -17756.042} C_VEL
LIN {X 0,Y 285.526,Z 233.064,A -85,B 0,C 180,E1 -17757.42,E2 -17757.42} C_VEL
LIN {X 0,Y 281.51,Z 208.081,A -85,B 0,C 180,E1 -17758.549,E2 -17758.549} C_VEL
LIN {X 0,Y 280.58,Z 204.469,A -85,B 0,C 180,E1 -17758.755,E2 -17758.755} C_VEL
LIN {X 0,Y 274.812,Z 190.815,A -85,B 0,C 180,E1 -17759.813,E2 -17759.813} C_VEL
LIN {X 0,Y 273.758,Z 187.904,A -85,B 0,C 180,E1 -17760.073,E2 -17760.073} C_VEL
LIN {X 0,Y 271.822,Z 178.857,A -85,B 0,C 180,E1 -17763.445,E2 -17763.445} C_VEL
LIN {X 0,Y 270.213,Z 172.328,A -85,B 0,C 180,E1 -17766.058,E2 -17766.058} C_VEL
LIN {X 0,Y 270.198,Z 172.33,A -85,B 0,C 180,E1 -17768.71,E2 -17768.71} C_VEL
LIN {X 0,Y 270.157,Z 172.334,A -85,B 0,C 180,E1 -17773.247,E2 -17773.247} C_VEL
LIN {X 0,Y 270.172,Z 172.33,A -85,B 0,C 180,E1 -17777.442,E2 -17777.442} C_VEL
LIN {X 0,Y 270.207,Z 172.326,A -85,B 0,C 180,E1 -17781.374,E2 -17781.374} C_VEL
LIN {X 0,Y 270.201,Z 172.326,A -85,B 0,C 180,E1 -17785.094,E2 -17785.094} C_VEL
LIN {X 0,Y 270.184,Z 172.328,A -85,B 0,C 180,E1 -17789.136,E2 -17789.136} C_VEL
LIN {X 0,Y 270.224,Z 172.322,A -85,B 0,C 180,E1 -17792.162,E2 -17792.162} C_VEL
LIN {X 0,Y 270.23,Z 172.324,A -85,B 0,C 180,E1 -17795.541,E2 -17795.541} C_VEL
LIN {X 0,Y 270.3,Z 172.314,A -85,B 0,C 180,E1 -17800.244,E2 -17800.244} C_VEL
LIN {X 0,Y 270.403,Z 172.301,A -85,B 0,C 180,E1 -17804.935,E2 -17804.935} C_VEL
LIN {X 0,Y 270.413,Z 172.301,A -85,B 0,C 180,E1 -17809.518,E2 -17809.518} C_VEL
LIN {X 0,Y 270.599,Z 172.273,A -85,B 0,C 180,E1 -17812.539,E2 -17812.539} C_VEL
LIN {X 0,Y 270.787,Z 172.25,A -85,B 0,C 180,E1 -17818.513,E2 -17818.513} C_VEL
LIN {X 0,Y 270.787,Z 172.255,A -85,B 0,C 180,E1 -17821.487,E2 -17821.487} C_VEL
LIN {X 0,Y 270.599,Z 172.277,A -85,B 0,C 180,E1 -17827.462,E2 -17827.462} C_VEL
LIN {X 0,Y 270.413,Z 172.3,A -85,B 0,C 180,E1 -17830.482,E2 -17830.482} C_VEL
LIN {X 0,Y 270.403,Z 172.302,A -85,B 0,C 180,E1 -17835.065,E2 -17835.065} C_VEL
LIN {X 0,Y 270.302,Z 172.313,A -85,B 0,C 180,E1 -17839.756,E2 -17839.756} C_VEL
LIN {X 0,Y 270.275,Z 172.32,A -85,B 0,C 180,E1 -17844.586,E2 -17844.586} C_VEL
LIN {X 0,Y 270.272,Z 172.313,A -85,B 0,C 180,E1 -17847.909,E2 -17847.909} C_VEL
LIN {X 0,Y 270.185,Z 172.326,A -85,B 0,C 180,E1 -17851.348,E2 -17851.348} C_VEL
LIN {X 0,Y 270.215,Z 172.323,A -85,B 0,C 180,E1 -17854.904,E2 -17854.904} C_VEL
LIN {X 0,Y 270.223,Z 172.322,A -85,B 0,C 180,E1 -17858.717,E2 -17858.717} C_VEL
LIN {X 0,Y 270.166,Z 172.329,A -85,B 0,C 180,E1 -17863.249,E2 -17863.249} C_VEL
LIN {X 0,Y 270.173,Z 172.331,A -85,B 0,C 180,E1 -17867.442,E2 -17867.442} C_VEL
LIN {X 0,Y 270.208,Z 172.328,A -85,B 0,C 180,E1 -17871.374,E2 -17871.374} C_VEL
LIN {X 0,Y 270.204,Z 172.331,A -85,B 0,C 180,E1 -17875.095,E2 -17875.095} C_VEL
LIN {X 0,Y 270.224,Z 172.349,A -85,B 0,C 180,E1 -17877.67,E2 -17877.67} C_VEL
LIN {X 0,Y 271.497,Z 177.583,A -85,B 0,C 180,E1 -17879.758,E2 -17879.758} C_VEL
LIN {X 0,Y 280.614,Z 197.623,A -85,B 0,C 180,E1 -17881.42,E2 -17881.42} C_VEL
LIN {X 0,Y 285.313,Z 209.778,A -85,B 0,C 180,E1 -17882.276,E2 -17882.276} C_VEL
LIN {X 0,Y 286.215,Z 215.199,A -85,B 0,C 180,E1 -17882.522,E2 -17882.522} C_VEL
LIN {X 0,Y 284.196,Z 282.877,A -85,B 0,C 180,E1 -17884.209,E2 -17884.209} C_VEL
LIN {X 0,Y 283.415,Z 295.374,A -85,B 0,C 180,E1 -17884.724,E2 -17884.724} C_VEL
LIN {X 0,Y 282.181,Z 308.168,A -85,B 0,C 180,E1 -17885.54,E2 -17885.54} C_VEL
LIN {X 0,Y 280.756,Z 320.013,A -85,B 0,C 180,E1 -17886.585,E2 -17886.585} C_VEL
LIN {X 0,Y 279.143,Z 330.764,A -85,B 0,C 180,E1 -17887.812,E2 -17887.812} C_VEL
LIN {X 0,Y 277.421,Z 340.648,A -85,B 0,C 180,E1 -17889.227,E2 -17889.227} C_VEL
LIN {X 0,Y 275.766,Z 350.616,A -85,B 0,C 180,E1 -17891.038,E2 -17891.038} C_VEL
LIN {X 0,Y 273.726,Z 360.264,A -85,B 0,C 180,E1 -17893.211,E2 -17893.211} C_VEL
LIN {X 0,Y 272.02,Z 367.956,A -85,B 0,C 180,E1 -17895.41,E2 -17895.41} C_VEL
LIN {X 0,Y 270.522,Z 375.015,A -85,B 0,C 180,E1 -17898.004,E2 -17898.004} C_VEL
LIN {X 0,Y 269.533,Z 379.716,A -85,B 0,C 180,E1 -17900.242,E2 -17900.242} C_VEL
LIN {X 0,Y 268.958,Z 383.31,A -85,B 0,C 180,E1 -17902.493,E2 -17902.493} C_VEL
LIN {X 0,Y 268.649,Z 385.167,A -85,B 0,C 180,E1 -17903.993,E2 -17903.993} C_VEL
LIN {X 0,Y 268.436,Z 386.564,A -85,B 0,C 180,E1 -17905.495,E2 -17905.495} C_VEL
LIN {X 0,Y 268.324,Z 387.557,A -85,B 0,C 180,E1 -17906.997,E2 -17906.997} C_VEL
LIN {X 0,Y 268.178,Z 388.399,A -85,B 0,C 180,E1 -17910,E2 -17910} C_VEL
LIN {X 0,Y 268.22,Z 388.206,A -85,B 0,C 180,E1 -17911.501,E2 -17911.501} C_VEL
LIN {X 0,Y 268.322,Z 387.619,A -85,B 0,C 180,E1 -17913.003,E2 -17913.003} C_VEL
LIN {X 0,Y 268.424,Z 386.652,A -85,B 0,C 180,E1 -17914.505,E2 -17914.505} C_VEL
LIN {X 0,Y 268.616,Z 385.131,A -85,B 0,C 180,E1 -17916.16,E2 -17916.16} C_VEL
LIN {X 0,Y 269.28,Z 381.227,A -85,B 0,C 180,E1 -17919.009,E2 -17919.009} C_VEL
LIN {X 0,Y 270.13,Z 376.97,A -85,B 0,C 180,E1 -17921.252,E2 -17921.252} C_VEL
LIN {X 0,Y 271.556,Z 370.522,A -85,B 0,C 180,E1 -17923.851,E2 -17923.851} C_VEL
LIN {X 0,Y 273.027,Z 363.436,A -85,B 0,C 180,E1 -17926.064,E2 -17926.064} C_VEL
LIN {X 0,Y 275.002,Z 354.605,A -85,B 0,C 180,E1 -17928.244,E2 -17928.244} C_VEL
LIN {X 0,Y 276.665,Z 345.335,A -85,B 0,C 180,E1 -17930.098,E2 -17930.098} C_VEL
LIN {X 0,Y 278.409,Z 335.509,A -85,B 0,C 180,E1 -17931.665,E2 -17931.665} C_VEL
LIN {X 0,Y 280.221,Z 324.34,A -85,B 0,C 180,E1 -17933.071,E2 -17933.071} C_VEL
LIN {X 0,Y 281.659,Z 313.786,A -85,B 0,C 180,E1 -17934.116,E2 -17934.116} C_VEL
LIN {X 0,Y 282.978,Z 301.067,A -85,B 0,C 180,E1 -17935.072,E2 -17935.072} C_VEL
LIN {X 0,Y 283.878,Z 289.482,A -85,B 0,C 180,E1 -17935.674,E2 -17935.674} C_VEL
LIN {X 0,Y 284.608,Z 273.906,A -85,B 0,C 180,E1 -17936.144,E2 -17936.144} C_VEL
LIN {X 0,Y 286.213,Z 214.511,A -85,B 0,C 180,E1 -17937.623,E2 -17937.623} C_VEL
LIN {X 0,Y 285.067,Z 209.027,A -85,B 0,C 180,E1 -17937.897,E2 -17937.897} C_VEL
LIN {X 0,Y 277.734,Z 190.793,A -85,B 0,C 180,E1 -17939.235,E2 -17939.235} C_VEL
LIN {X 0,Y 271.458,Z 177.344,A -85,B 0,C 180,E1 -17940.432,E2 -17940.432} C_VEL
LIN {X 0,Y 270.227,Z 172.326,A -85,B 0,C 180,E1 -17942.55,E2 -17942.55} C_VEL
LIN {X 0,Y 270.218,Z 172.325,A -85,B 0,C 180,E1 -17946.741,E2 -17946.741} C_VEL
LIN {X 0,Y 270.17,Z 172.331,A -85,B 0,C 180,E1 -17951.028,E2 -17951.028} C_VEL
LIN {X 0,Y 270.153,Z 172.33,A -85,B 0,C 180,E1 -17955.38,E2 -17955.38} C_VEL
LIN {X 0,Y 270.174,Z 172.328,A -85,B 0,C 180,E1 -17959.434,E2 -17959.434} C_VEL
LIN {X 0,Y 270.229,Z 172.32,A -85,B 0,C 180,E1 -17963.261,E2 -17963.261} C_VEL
LIN {X 0,Y 270.203,Z 172.318,A -85,B 0,C 180,E1 -17966.892,E2 -17966.892} C_VEL
LIN {X 0,Y 270.229,Z 172.32,A -85,B 0,C 180,E1 -17970.386,E2 -17970.386} C_VEL
LIN {X 0,Y 270.264,Z 172.32,A -85,B 0,C 180,E1 -17973.764,E2 -17973.764} C_VEL
LIN {X 0,Y 270.233,Z 172.32,A -85,B 0,C 180,E1 -17977.039,E2 -17977.039} C_VEL
LIN {X 0,Y 270.302,Z 172.313,A -85,B 0,C 180,E1 -17980.244,E2 -17980.244} C_VEL
LIN {X 0,Y 270.403,Z 172.293,A -85,B 0,C 180,E1 -17984.935,E2 -17984.935} C_VEL
LIN {X 0,Y 270.364,Z 172.297,A -85,B 0,C 180,E1 -17985.506,E2 -17985.506} C_VEL
LIN {X 0,Y 269.679,Z 172.391,A -85,B 0,C 180,E1 -17986.749,E2 -17986.749} C_VEL
LIN {X 0,Y 266.888,Z 172.74,A -85,B 0,C 180,E1 -17988.778,E2 -17988.778} C_VEL
LIN {X 0,Y 264.568,Z 173.023,A -85,B 0,C 180,E1 -17990.428,E2 -17990.428} C_VEL
LIN {X 0,Y 263.614,Z 173.138,A -85,B 0,C 180,E1 -17991.704,E2 -17991.704} C_VEL
LIN {X 0,Y 263.557,Z 173.144,A -85,B 0,C 180,E1 -17992.136,E2 -17992.136} C_VEL
LIN {X 0,Y 263.564,Z 173.15,A -85,B 0,C 180,E1 -17996.943,E2 -17996.943} C_VEL
LIN {X 0,Y 263.795,Z 173.118,A -85,B 0,C 180,E1 -18000,E2 -18000} C_VEL
LIN {X 0,Y 263.563,Z 173.154,A -85,B 0,C 180,E1 -18003.057,E2 -18003.057} C_VEL
LIN {X 0,Y 263.569,Z 173.148,A -85,B 0,C 180,E1 -18007.662,E2 -18007.662} C_VEL
LIN {X 0,Y 263.373,Z 173.176,A -85,B 0,C 180,E1 -18010.766,E2 -18010.766} C_VEL
LIN {X 0,Y 263.35,Z 173.177,A -85,B 0,C 180,E1 -18015.478,E2 -18015.478} C_VEL
LIN {X 0,Y 263.262,Z 173.185,A -85,B 0,C 180,E1 -18020.307,E2 -18020.307} C_VEL
LIN {X 0,Y 263.192,Z 173.192,A -85,B 0,C 180,E1 -18025.293,E2 -18025.293} C_VEL
LIN {X 0,Y 263.165,Z 173.201,A -85,B 0,C 180,E1 -18028.731,E2 -18028.731} C_VEL
LIN {X 0,Y 263.132,Z 173.208,A -85,B 0,C 180,E1 -18032.288,E2 -18032.288} C_VEL
LIN {X 0,Y 263.181,Z 173.201,A -85,B 0,C 180,E1 -18036.763,E2 -18036.763} C_VEL
LIN {X 0,Y 263.124,Z 173.207,A -85,B 0,C 180,E1 -18041.594,E2 -18041.594} C_VEL
LIN {X 0,Y 263.101,Z 173.211,A -85,B 0,C 180,E1 -18046.012,E2 -18046.012} C_VEL
LIN {X 0,Y 263.091,Z 173.212,A -85,B 0,C 180,E1 -18050.125,E2 -18050.125} C_VEL
LIN {X 0,Y 263.18,Z 173.255,A -85,B 0,C 180,E1 -18053.238,E2 -18053.238} C_VEL
LIN {X 0,Y 265.5,Z 182.849,A -85,B 0,C 180,E1 -18057.117,E2 -18057.117} C_VEL
LIN {X 0,Y 266.577,Z 187.891,A -85,B 0,C 180,E1 -18059.041,E2 -18059.041} C_VEL
LIN {X 0,Y 274.389,Z 206.502,A -85,B 0,C 180,E1 -18060.558,E2 -18060.558} C_VEL
LIN {X 0,Y 275.359,Z 209.641,A -85,B 0,C 180,E1 -18060.763,E2 -18060.763} C_VEL
LIN {X 0,Y 278.765,Z 230.175,A -85,B 0,C 180,E1 -18061.741,E2 -18061.741} C_VEL
LIN {X 0,Y 279.383,Z 235.703,A -85,B 0,C 180,E1 -18061.967,E2 -18061.967} C_VEL
LIN {X 0,Y 277.435,Z 296.563,A -85,B 0,C 180,E1 -18063.533,E2 -18063.533} C_VEL
LIN {X 0,Y 276.453,Z 308.938,A -85,B 0,C 180,E1 -18064.091,E2 -18064.091} C_VEL
LIN {X 0,Y 275.064,Z 321.791,A -85,B 0,C 180,E1 -18064.965,E2 -18064.965} C_VEL
LIN {X 0,Y 273.317,Z 333.998,A -85,B 0,C 180,E1 -18066.11,E2 -18066.11} C_VEL
LIN {X 0,Y 271.333,Z 345.561,A -85,B 0,C 180,E1 -18067.539,E2 -18067.539} C_VEL
LIN {X 0,Y 269.264,Z 355.974,A -85,B 0,C 180,E1 -18069.169,E2 -18069.169} C_VEL
LIN {X 0,Y 267.592,Z 364.435,A -85,B 0,C 180,E1 -18070.822,E2 -18070.822} C_VEL
LIN {X 0,Y 265.979,Z 372.352,A -85,B 0,C 180,E1 -18072.707,E2 -18072.707} C_VEL
LIN {X 0,Y 264.279,Z 380.027,A -85,B 0,C 180,E1 -18074.973,E2 -18074.973} C_VEL
LIN {X 0,Y 262.752,Z 387.108,A -85,B 0,C 180,E1 -18077.644,E2 -18077.644} C_VEL
LIN {X 0,Y 261.914,Z 391.822,A -85,B 0,C 180,E1 -18079.955,E2 -18079.955} C_VEL
LIN {X 0,Y 261.352,Z 395.423,A -85,B 0,C 180,E1 -18082.273,E2 -18082.273} C_VEL
LIN {X 0,Y 261.024,Z 398.409,A -85,B 0,C 180,E1 -18085.015,E2 -18085.015} C_VEL
LIN {X 0,Y 261.048,Z 399.671,A -85,B 0,C 180,E1 -18086.914,E2 -18086.914} C_VEL
LIN {X 0,Y 261.08,Z 400.279,A -85,B 0,C 180,E1 -18088.458,E2 -18088.458} C_VEL
LIN {X 0,Y 261.099,Z 400.491,A -85,B 0,C 180,E1 -18090,E2 -18090} C_VEL
LIN {X 0,Y 261.08,Z 400.269,A -85,B 0,C 180,E1 -18091.543,E2 -18091.543} C_VEL
LIN {X 0,Y 261.048,Z 399.655,A -85,B 0,C 180,E1 -18093.087,E2 -18093.087} C_VEL
LIN {X 0,Y 261.085,Z 398.243,A -85,B 0,C 180,E1 -18095.137,E2 -18095.137} C_VEL
LIN {X 0,Y 261.352,Z 395.379,A -85,B 0,C 180,E1 -18097.727,E2 -18097.727} C_VEL
LIN {X 0,Y 261.914,Z 391.758,A -85,B 0,C 180,E1 -18100.045,E2 -18100.045} C_VEL
LIN {X 0,Y 262.751,Z 387.028,A -85,B 0,C 180,E1 -18102.356,E2 -18102.356} C_VEL
LIN {X 0,Y 264.285,Z 379.929,A -85,B 0,C 180,E1 -18105.027,E2 -18105.027} C_VEL
LIN {X 0,Y 265.955,Z 372.221,A -85,B 0,C 180,E1 -18107.295,E2 -18107.295} C_VEL
LIN {X 0,Y 267.877,Z 362.546,A -85,B 0,C 180,E1 -18109.542,E2 -18109.542} C_VEL
LIN {X 0,Y 269.879,Z 352.564,A -85,B 0,C 180,E1 -18111.382,E2 -18111.382} C_VEL
LIN {X 0,Y 271.994,Z 341.286,A -85,B 0,C 180,E1 -18113.005,E2 -18113.005} C_VEL
LIN {X 0,Y 273.777,Z 330.235,A -85,B 0,C 180,E1 -18114.251,E2 -18114.251} C_VEL
LIN {X 0,Y 275.435,Z 317.975,A -85,B 0,C 180,E1 -18115.302,E2 -18115.302} C_VEL
LIN {X 0,Y 276.727,Z 305.954,A -85,B 0,C 180,E1 -18116.033,E2 -18116.033} C_VEL
LIN {X 0,Y 277.644,Z 292.746,A -85,B 0,C 180,E1 -18116.547,E2 -18116.547} C_VEL
LIN {X 0,Y 279.238,Z 234.053,A -85,B 0,C 180,E1 -18118.058,E2 -18118.058} C_VEL
LIN {X 0,Y 275.375,Z 209.764,A -85,B 0,C 180,E1 -18119.192,E2 -18119.192} C_VEL
LIN {X 0,Y 274.319,Z 206.292,A -85,B 0,C 180,E1 -18119.416,E2 -18119.416} C_VEL
LIN {X 0,Y 267.809,Z 190.967,A -85,B 0,C 180,E1 -18120.664,E2 -18120.664} C_VEL
LIN {X 0,Y 266.541,Z 187.817,A -85,B 0,C 180,E1 -18120.938,E2 -18120.938} C_VEL
LIN {X 0,Y 264.5,Z 178.539,A -85,B 0,C 180,E1 -18124.543,E2 -18124.543} C_VEL
LIN {X 0,Y 263.179,Z 173.204,A -85,B 0,C 180,E1 -18126.762,E2 -18126.762} C_VEL
LIN {X 0,Y 263.091,Z 173.214,A -85,B 0,C 180,E1 -18129.875,E2 -18129.875} C_VEL
LIN {X 0,Y 263.102,Z 173.213,A -85,B 0,C 180,E1 -18133.988,E2 -18133.988} C_VEL
LIN {X 0,Y 263.124,Z 173.211,A -85,B 0,C 180,E1 -18138.406,E2 -18138.406} C_VEL
LIN {X 0,Y 263.182,Z 173.201,A -85,B 0,C 180,E1 -18143.237,E2 -18143.237} C_VEL
LIN {X 0,Y 263.128,Z 173.208,A -85,B 0,C 180,E1 -18147.711,E2 -18147.711} C_VEL
LIN {X 0,Y 263.151,Z 173.206,A -85,B 0,C 180,E1 -18151.803,E2 -18151.803} C_VEL
LIN {X 0,Y 263.193,Z 173.199,A -85,B 0,C 180,E1 -18155.216,E2 -18155.216} C_VEL
LIN {X 0,Y 263.262,Z 173.193,A -85,B 0,C 180,E1 -18159.693,E2 -18159.693} C_VEL
LIN {X 0,Y 263.351,Z 173.179,A -85,B 0,C 180,E1 -18164.522,E2 -18164.522} C_VEL
LIN {X 0,Y 263.355,Z 173.177,A -85,B 0,C 180,E1 -18169.234,E2 -18169.234} C_VEL
LIN {X 0,Y 263.558,Z 173.15,A -85,B 0,C 180,E1 -18172.338,E2 -18172.338} C_VEL
LIN {X 0,Y 263.752,Z 173.127,A -85,B 0,C 180,E1 -18178.473,E2 -18178.473} C_VEL
LIN {X 0,Y 263.751,Z 173.131,A -85,B 0,C 180,E1 -18181.527,E2 -18181.527} C_VEL
LIN {X 0,Y 263.558,Z 173.154,A -85,B 0,C 180,E1 -18187.662,E2 -18187.662} C_VEL
LIN {X 0,Y 263.355,Z 173.176,A -85,B 0,C 180,E1 -18190.766,E2 -18190.766} C_VEL
LIN {X 0,Y 263.351,Z 173.178,A -85,B 0,C 180,E1 -18195.478,E2 -18195.478} C_VEL
LIN {X 0,Y 263.264,Z 173.192,A -85,B 0,C 180,E1 -18200.307,E2 -18200.307} C_VEL
LIN {X 0,Y 263.209,Z 173.197,A -85,B 0,C 180,E1 -18205.291,E2 -18205.291} C_VEL
LIN {X 0,Y 263.18,Z 173.202,A -85,B 0,C 180,E1 -18208.73,E2 -18208.73} C_VEL
LIN {X 0,Y 263.134,Z 173.205,A -85,B 0,C 180,E1 -18212.288,E2 -18212.288} C_VEL
LIN {X 0,Y 263.188,Z 173.199,A -85,B 0,C 180,E1 -18215.978,E2 -18215.978} C_VEL
LIN {X 0,Y 263.116,Z 173.208,A -85,B 0,C 180,E1 -18219.871,E2 -18219.871} C_VEL
LIN {X 0,Y 263.123,Z 173.21,A -85,B 0,C 180,E1 -18223.984,E2 -18223.984} C_VEL
LIN {X 0,Y 263.125,Z 173.208,A -85,B 0,C 180,E1 -18228.407,E2 -18228.407} C_VEL
LIN {X 0,Y 263.186,Z 173.204,A -85,B 0,C 180,E1 -18233.236,E2 -18233.236} C_VEL
LIN {X 0,Y 263.174,Z 173.263,A -85,B 0,C 180,E1 -18236.979,E2 -18236.979} C_VEL
LIN {X 0,Y 264.266,Z 177.715,A -85,B 0,C 180,E1 -18238.837,E2 -18238.837} C_VEL
LIN {X 0,Y 273.08,Z 196.533,A -85,B 0,C 180,E1 -18240.516,E2 -18240.516} C_VEL
LIN {X 0,Y 279.076,Z 211.743,A -85,B 0,C 180,E1 -18241.652,E2 -18241.652} C_VEL
LIN {X 0,Y 279.942,Z 215.985,A -85,B 0,C 180,E1 -18241.87,E2 -18241.87} C_VEL
LIN {X 0,Y 277.836,Z 283.059,A -85,B 0,C 180,E1 -18243.574,E2 -18243.574} C_VEL
LIN {X 0,Y 277.028,Z 295.547,A -85,B 0,C 180,E1 -18244.098,E2 -18244.098} C_VEL
LIN {X 0,Y 275.746,Z 308.337,A -85,B 0,C 180,E1 -18244.93,E2 -18244.93} C_VEL
LIN {X 0,Y 274.263,Z 320.181,A -85,B 0,C 180,E1 -18245.996,E2 -18245.996} C_VEL
LIN {X 0,Y 272.574,Z 330.931,A -85,B 0,C 180,E1 -18247.247,E2 -18247.247} C_VEL
LIN {X 0,Y 270.808,Z 340.813,A -85,B 0,C 180,E1 -18248.695,E2 -18248.695} C_VEL
LIN {X 0,Y 269.052,Z 350.781,A -85,B 0,C 180,E1 -18250.546,E2 -18250.546} C_VEL
LIN {X 0,Y 266.94,Z 360.428,A -85,B 0,C 180,E1 -18252.771,E2 -18252.771} C_VEL
LIN {X 0,Y 265.124,Z 368.12,A -85,B 0,C 180,E1 -18255.022,E2 -18255.022} C_VEL
LIN {X 0,Y 263.584,Z 375.178,A -85,B 0,C 180,E1 -18257.684,E2 -18257.684} C_VEL
LIN {X 0,Y 262.525,Z 379.88,A -85,B 0,C 180,E1 -18259.979,E2 -18259.979} C_VEL
LIN {X 0,Y 261.899,Z 383.474,A -85,B 0,C 180,E1 -18262.289,E2 -18262.289} C_VEL
LIN {X 0,Y 261.592,Z 385.33,A -85,B 0,C 180,E1 -18263.831,E2 -18263.831} C_VEL
LIN {X 0,Y 261.353,Z 386.727,A -85,B 0,C 180,E1 -18265.373,E2 -18265.373} C_VEL
LIN {X 0,Y 261.24,Z 387.719,A -85,B 0,C 180,E1 -18266.916,E2 -18266.916} C_VEL
LIN {X 0,Y 261.15,Z 388.33,A -85,B 0,C 180,E1 -18268.458,E2 -18268.458} C_VEL
LIN {X 0,Y 261.105,Z 388.561,A -85,B 0,C 180,E1 -18270,E2 -18270} C_VEL
LIN {X 0,Y 261.15,Z 388.368,A -85,B 0,C 180,E1 -18271.542,E2 -18271.542} C_VEL
LIN {X 0,Y 261.237,Z 387.781,A -85,B 0,C 180,E1 -18273.084,E2 -18273.084} C_VEL
LIN {X 0,Y 261.518,Z 385.456,A -85,B 0,C 180,E1 -18276.171,E2 -18276.171} C_VEL
LIN {X 0,Y 262.038,Z 382.585,A -85,B 0,C 180,E1 -18278.483,E2 -18278.483} C_VEL
LIN {X 0,Y 262.829,Z 378.691,A -85,B 0,C 180,E1 -18280.788,E2 -18280.788} C_VEL
LIN {X 0,Y 263.927,Z 373.668,A -85,B 0,C 180,E1 -18283.082,E2 -18283.082} C_VEL
LIN {X 0,Y 265.317,Z 367.341,A -85,B 0,C 180,E1 -18285.36,E2 -18285.36} C_VEL
LIN {X 0,Y 267.207,Z 359.42,A -85,B 0,C 180,E1 -18287.606,E2 -18287.606} C_VEL
LIN {X 0,Y 268.907,Z 351.347,A -85,B 0,C 180,E1 -18289.465,E2 -18289.465} C_VEL
LIN {X 0,Y 270.761,Z 341.497,A -85,B 0,C 180,E1 -18291.308,E2 -18291.308} C_VEL
LIN {X 0,Y 272.715,Z 330.407,A -85,B 0,C 180,E1 -18292.941,E2 -18292.941} C_VEL
LIN {X 0,Y 274.438,Z 319.531,A -85,B 0,C 180,E1 -18294.188,E2 -18294.188} C_VEL
LIN {X 0,Y 275.966,Z 307.513,A -85,B 0,C 180,E1 -18295.25,E2 -18295.25} C_VEL
LIN {X 0,Y 277.058,Z 295.16,A -85,B 0,C 180,E1 -18296.05,E2 -18296.05} C_VEL
LIN {X 0,Y 277.946,Z 282.339,A -85,B 0,C 180,E1 -18296.566,E2 -18296.566} C_VEL
LIN {X 0,Y 279.96,Z 215.762,A -85,B 0,C 180,E1 -18298.263,E2 -18298.263} C_VEL
LIN {X 0,Y 279.142,Z 211.757,A -85,B 0,C 180,E1 -18298.469,E2 -18298.469} C_VEL
LIN {X 0,Y 272.06,Z 194.092,A -85,B 0,C 180,E1 -18299.811,E2 -18299.811} C_VEL
LIN {X 0,Y 265.378,Z 180.273,A -85,B 0,C 180,E1 -18301.073,E2 -18301.073} C_VEL
LIN {X 0,Y 264.231,Z 177.529,A -85,B 0,C 180,E1 -18301.358,E2 -18301.358} C_VEL
LIN {X 0,Y 263.169,Z 173.205,A -85,B 0,C 180,E1 -18303.193,E2 -18303.193} C_VEL
LIN {X 0,Y 263.184,Z 173.201,A -85,B 0,C 180,E1 -18306.763,E2 -18306.763} C_VEL
LIN {X 0,Y 263.125,Z 173.208,A -85,B 0,C 180,E1 -18311.593,E2 -18311.593} C_VEL
LIN {X 0,Y 263.123,Z 173.209,A -85,B 0,C 180,E1 -18316.016,E2 -18316.016} C_VEL
LIN {X 0,Y 263.116,Z 173.211,A -85,B 0,C 180,E1 -18320.129,E2 -18320.129} C_VEL
LIN {X 0,Y 263.177,Z 173.203,A -85,B 0,C 180,E1 -18324.02,E2 -18324.02} C_VEL
LIN {X 0,Y 263.133,Z 173.203,A -85,B 0,C 180,E1 -18327.712,E2 -18327.712} C_VEL
LIN {X 0,Y 263.201,Z 173.192,A -85,B 0,C 180,E1 -18331.783,E2 -18331.783} C_VEL
LIN {X 0,Y 263.226,Z 173.197,A -85,B 0,C 180,E1 -18335.2,E2 -18335.2} C_VEL
LIN {X 0,Y 263.264,Z 173.191,A -85,B 0,C 180,E1 -18339.693,E2 -18339.693} C_VEL
LIN {X 0,Y 263.351,Z 173.169,A -85,B 0,C 180,E1 -18344.522,E2 -18344.522} C_VEL
LIN {X 0,Y 263.374,Z 173.176,A -85,B 0,C 180,E1 -18349.234,E2 -18349.234} C_VEL
LIN {X 0,Y 263.557,Z 173.144,A -85,B 0,C 180,E1 -18352.136,E2 -18352.136} C_VEL
LIN {X 0,Y 262.956,Z 173.229,A -85,B 0,C 180,E1 -18353.409,E2 -18353.409} C_VEL
LIN {X 0,Y 260.183,Z 173.574,A -85,B 0,C 180,E1 -18355.487,E2 -18355.487} C_VEL
LIN {X 0,Y 257.801,Z 173.866,A -85,B 0,C 180,E1 -18357.177,E2 -18357.177} C_VEL
LIN {X 0,Y 256.785,Z 173.988,A -85,B 0,C 180,E1 -18358.486,E2 -18358.486} C_VEL
LIN {X 0,Y 256.707,Z 173.996,A -85,B 0,C 180,E1 -18358.929,E2 -18358.929} C_VEL
LIN {X 0,Y 256.714,Z 174.006,A -85,B 0,C 180,E1 -18361.569,E2 -18361.569} C_VEL
LIN {X 0,Y 256.537,Z 174.024,A -85,B 0,C 180,E1 -18367.873,E2 -18367.873} C_VEL
LIN {X 0,Y 256.309,Z 174.054,A -85,B 0,C 180,E1 -18371.066,E2 -18371.066} C_VEL
LIN {X 0,Y 256.299,Z 174.057,A -85,B 0,C 180,E1 -18375.915,E2 -18375.915} C_VEL
LIN {X 0,Y 256.162,Z 174.073,A -85,B 0,C 180,E1 -18380.896,E2 -18380.896} C_VEL
LIN {X 0,Y 256.17,Z 174.066,A -85,B 0,C 180,E1 -18385.13,E2 -18385.13} C_VEL
LIN {X 0,Y 256.103,Z 174.08,A -85,B 0,C 180,E1 -18389.601,E2 -18389.601} C_VEL
LIN {X 0,Y 256.067,Z 174.088,A -85,B 0,C 180,E1 -18393.293,E2 -18393.293} C_VEL
LIN {X 0,Y 256.114,Z 174.083,A -85,B 0,C 180,E1 -18397.271,E2 -18397.271} C_VEL
LIN {X 0,Y 256.054,Z 174.088,A -85,B 0,C 180,E1 -18401.204,E2 -18401.204} C_VEL
LIN {X 0,Y 256.039,Z 174.093,A -85,B 0,C 180,E1 -18405.535,E2 -18405.535} C_VEL
LIN {X 0,Y 256.04,Z 174.091,A -85,B 0,C 180,E1 -18408.794,E2 -18408.794} C_VEL
LIN {X 0,Y 256.131,Z 174.178,A -85,B 0,C 180,E1 -18412.492,E2 -18412.492} C_VEL
LIN {X 0,Y 258.247,Z 182.71,A -85,B 0,C 180,E1 -18416.09,E2 -18416.09} C_VEL
LIN {X 0,Y 259.355,Z 187.7,A -85,B 0,C 180,E1 -18418.078,E2 -18418.078} C_VEL
LIN {X 0,Y 267.647,Z 207.027,A -85,B 0,C 180,E1 -18419.761,E2 -18419.761} C_VEL
LIN {X 0,Y 269.334,Z 211.714,A -85,B 0,C 180,E1 -18420.11,E2 -18420.11} C_VEL
LIN {X 0,Y 272.649,Z 232.272,A -85,B 0,C 180,E1 -18421.114,E2 -18421.114} C_VEL
LIN {X 0,Y 273.058,Z 238.143,A -85,B 0,C 180,E1 -18421.333,E2 -18421.333} C_VEL
LIN {X 0,Y 271.116,Z 296.415,A -85,B 0,C 180,E1 -18422.866,E2 -18422.866} C_VEL
LIN {X 0,Y 270.006,Z 309.548,A -85,B 0,C 180,E1 -18423.477,E2 -18423.477} C_VEL
LIN {X 0,Y 268.658,Z 321.636,A -85,B 0,C 180,E1 -18424.325,E2 -18424.325} C_VEL
LIN {X 0,Y 266.835,Z 333.84,A -85,B 0,C 180,E1 -18425.492,E2 -18425.492} C_VEL
LIN {X 0,Y 264.783,Z 345.403,A -85,B 0,C 180,E1 -18426.952,E2 -18426.952} C_VEL
LIN {X 0,Y 262.619,Z 355.815,A -85,B 0,C 180,E1 -18428.616,E2 -18428.616} C_VEL
LIN {X 0,Y 260.586,Z 365.554,A -85,B 0,C 180,E1 -18430.596,E2 -18430.596} C_VEL
LIN {X 0,Y 258.85,Z 373.565,A -85,B 0,C 180,E1 -18432.623,E2 -18432.623} C_VEL
LIN {X 0,Y 257.14,Z 380.986,A -85,B 0,C 180,E1 -18434.951,E2 -18434.951} C_VEL
LIN {X 0,Y 255.779,Z 386.946,A -85,B 0,C 180,E1 -18437.302,E2 -18437.302} C_VEL
LIN {X 0,Y 254.886,Z 391.659,A -85,B 0,C 180,E1 -18439.675,E2 -18439.675} C_VEL
LIN {X 0,Y 254.311,Z 395.261,A -85,B 0,C 180,E1 -18442.058,E2 -18442.058} C_VEL
LIN {X 0,Y 253.952,Z 398.385,A -85,B 0,C 180,E1 -18445.059,E2 -18445.059} C_VEL
LIN {X 0,Y 253.947,Z 399.509,A -85,B 0,C 180,E1 -18446.827,E2 -18446.827} C_VEL
LIN {X 0,Y 253.987,Z 400.117,A -85,B 0,C 180,E1 -18448.414,E2 -18448.414} C_VEL
LIN {X 0,Y 254.027,Z 400.329,A -85,B 0,C 180,E1 -18450,E2 -18450} C_VEL
LIN {X 0,Y 253.987,Z 400.106,A -85,B 0,C 180,E1 -18451.586,E2 -18451.586} C_VEL
LIN {X 0,Y 253.947,Z 399.493,A -85,B 0,C 180,E1 -18453.173,E2 -18453.173} C_VEL
LIN {X 0,Y 253.99,Z 398.291,A -85,B 0,C 180,E1 -18455.039,E2 -18455.039} C_VEL
LIN {X 0,Y 254.312,Z 395.216,A -85,B 0,C 180,E1 -18457.942,E2 -18457.942} C_VEL
LIN {X 0,Y 254.886,Z 391.594,A -85,B 0,C 180,E1 -18460.325,E2 -18460.325} C_VEL
LIN {X 0,Y 255.777,Z 386.863,A -85,B 0,C 180,E1 -18462.698,E2 -18462.698} C_VEL
LIN {X 0,Y 257.421,Z 379.765,A -85,B 0,C 180,E1 -18465.438,E2 -18465.438} C_VEL
LIN {X 0,Y 259.145,Z 372.175,A -85,B 0,C 180,E1 -18467.731,E2 -18467.731} C_VEL
LIN {X 0,Y 260.788,Z 364.169,A -85,B 0,C 180,E1 -18469.685,E2 -18469.685} C_VEL
LIN {X 0,Y 262.821,Z 354.542,A -85,B 0,C 180,E1 -18471.573,E2 -18471.573} C_VEL
LIN {X 0,Y 264.975,Z 343.867,A -85,B 0,C 180,E1 -18473.237,E2 -18473.237} C_VEL
LIN {X 0,Y 266.77,Z 333.543,A -85,B 0,C 180,E1 -18474.515,E2 -18474.515} C_VEL
LIN {X 0,Y 268.571,Z 321.199,A -85,B 0,C 180,E1 -18475.684,E2 -18475.684} C_VEL
LIN {X 0,Y 270.112,Z 308.198,A -85,B 0,C 180,E1 -18476.564,E2 -18476.564} C_VEL
LIN {X 0,Y 271.169,Z 295.521,A -85,B 0,C 180,E1 -18477.128,E2 -18477.128} C_VEL
LIN {X 0,Y 272.972,Z 234.973,A -85,B 0,C 180,E1 -18478.729,E2 -18478.729} C_VEL
LIN {X 0,Y 269.18,Z 210.92,A -85,B 0,C 180,E1 -18479.891,E2 -18479.891} C_VEL
LIN {X 0,Y 263.711,Z 197.74,A -85,B 0,C 180,E1 -18480.979,E2 -18480.979} C_VEL
LIN {X 0,Y 259.305,Z 187.607,A -85,B 0,C 180,E1 -18481.907,E2 -18481.907} C_VEL
LIN {X 0,Y 257.285,Z 178.796,A -85,B 0,C 180,E1 -18485.482,E2 -18485.482} C_VEL
LIN {X 0,Y 256.128,Z 174.082,A -85,B 0,C 180,E1 -18487.507,E2 -18487.507} C_VEL
LIN {X 0,Y 256.059,Z 174.09,A -85,B 0,C 180,E1 -18492.178,E2 -18492.178} C_VEL
LIN {X 0,Y 256.049,Z 174.093,A -85,B 0,C 180,E1 -18496.67,E2 -18496.67} C_VEL
LIN {X 0,Y 256.071,Z 174.088,A -85,B 0,C 180,E1 -18500.858,E2 -18500.858} C_VEL
LIN {X 0,Y 256.13,Z 174.08,A -85,B 0,C 180,E1 -18502.867,E2 -18502.867} C_VEL
LIN {X 0,Y 256.066,Z 174.088,A -85,B 0,C 180,E1 -18506.707,E2 -18506.707} C_VEL
LIN {X 0,Y 256.056,Z 174.091,A -85,B 0,C 180,E1 -18510.393,E2 -18510.393} C_VEL
LIN {X 0,Y 256.161,Z 174.075,A -85,B 0,C 180,E1 -18514.875,E2 -18514.875} C_VEL
LIN {X 0,Y 256.162,Z 174.074,A -85,B 0,C 180,E1 -18519.104,E2 -18519.104} C_VEL
LIN {X 0,Y 256.3,Z 174.059,A -85,B 0,C 180,E1 -18524.085,E2 -18524.085} C_VEL
LIN {X 0,Y 256.298,Z 174.055,A -85,B 0,C 180,E1 -18528.933,E2 -18528.933} C_VEL
LIN {X 0,Y 256.515,Z 174.028,A -85,B 0,C 180,E1 -18532.126,E2 -18532.126} C_VEL
LIN {X 0,Y 256.499,Z 174.034,A -85,B 0,C 180,E1 -18536.859,E2 -18536.859} C_VEL
LIN {X 0,Y 256.758,Z 173.996,A -85,B 0,C 180,E1 -18540,E2 -18540} C_VEL
LIN {X 0,Y 256.498,Z 174.035,A -85,B 0,C 180,E1 -18543.141,E2 -18543.141} C_VEL
LIN {X 0,Y 256.515,Z 174.031,A -85,B 0,C 180,E1 -18547.874,E2 -18547.874} C_VEL
LIN {X 0,Y 256.295,Z 174.054,A -85,B 0,C 180,E1 -18552.672,E2 -18552.672} C_VEL
LIN {X 0,Y 256.283,Z 174.059,A -85,B 0,C 180,E1 -18556.302,E2 -18556.302} C_VEL
LIN {X 0,Y 256.158,Z 174.074,A -85,B 0,C 180,E1 -18561.12,E2 -18561.12} C_VEL
LIN {X 0,Y 256.189,Z 174.072,A -85,B 0,C 180,E1 -18565.139,E2 -18565.139} C_VEL
LIN {X 0,Y 256.115,Z 174.081,A -85,B 0,C 180,E1 -18569.6,E2 -18569.6} C_VEL
LIN {X 0,Y 256.086,Z 174.084,A -85,B 0,C 180,E1 -18573.29,E2 -18573.29} C_VEL
LIN {X 0,Y 256.129,Z 174.079,A -85,B 0,C 180,E1 -18577.275,E2 -18577.275} C_VEL
LIN {X 0,Y 256.057,Z 174.089,A -85,B 0,C 180,E1 -18581.203,E2 -18581.203} C_VEL
LIN {X 0,Y 256.058,Z 174.086,A -85,B 0,C 180,E1 -18585.53,E2 -18585.53} C_VEL
LIN {X 0,Y 256.056,Z 174.088,A -85,B 0,C 180,E1 -18588.797,E2 -18588.797} C_VEL
LIN {X 0,Y 256.133,Z 174.081,A -85,B 0,C 180,E1 -18592.868,E2 -18592.868} C_VEL
LIN {X 0,Y 256.162,Z 174.262,A -85,B 0,C 180,E1 -18596.283,E2 -18596.283} C_VEL
LIN {X 0,Y 257.058,Z 177.973,A -85,B 0,C 180,E1 -18597.861,E2 -18597.861} C_VEL
LIN {X 0,Y 265.734,Z 195.962,A -85,B 0,C 180,E1 -18599.592,E2 -18599.592} C_VEL
LIN {X 0,Y 271.942,Z 210.997,A -85,B 0,C 180,E1 -18600.81,E2 -18600.81} C_VEL
LIN {X 0,Y 273.563,Z 216.055,A -85,B 0,C 180,E1 -18601.149,E2 -18601.149} C_VEL
LIN {X 0,Y 271.591,Z 281.738,A -85,B 0,C 180,E1 -18602.865,E2 -18602.865} C_VEL
LIN {X 0,Y 270.732,Z 294.857,A -85,B 0,C 180,E1 -18603.398,E2 -18603.398} C_VEL
LIN {X 0,Y 269.475,Z 307.379,A -85,B 0,C 180,E1 -18604.201,E2 -18604.201} C_VEL
LIN {X 0,Y 267.805,Z 320.349,A -85,B 0,C 180,E1 -18605.379,E2 -18605.379} C_VEL
LIN {X 0,Y 266.046,Z 331.098,A -85,B 0,C 180,E1 -18606.656,E2 -18606.656} C_VEL
LIN {X 0,Y 263.994,Z 342.04,A -85,B 0,C 180,E1 -18608.32,E2 -18608.32} C_VEL
LIN {X 0,Y 262.349,Z 350.947,A -85,B 0,C 180,E1 -18610.028,E2 -18610.028} C_VEL
LIN {X 0,Y 260.492,Z 359.113,A -85,B 0,C 180,E1 -18611.925,E2 -18611.925} C_VEL
LIN {X 0,Y 258.534,Z 367.116,A -85,B 0,C 180,E1 -18614.226,E2 -18614.226} C_VEL
LIN {X 0,Y 257.048,Z 373.534,A -85,B 0,C 180,E1 -18616.562,E2 -18616.562} C_VEL
LIN {X 0,Y 255.858,Z 378.625,A -85,B 0,C 180,E1 -18618.914,E2 -18618.914} C_VEL
LIN {X 0,Y 255.038,Z 382.576,A -85,B 0,C 180,E1 -18621.283,E2 -18621.283} C_VEL
LIN {X 0,Y 254.506,Z 385.619,A -85,B 0,C 180,E1 -18623.784,E2 -18623.784} C_VEL
LIN {X 0,Y 254.158,Z 387.881,A -85,B 0,C 180,E1 -18626.83,E2 -18626.83} C_VEL
LIN {X 0,Y 254.035,Z 388.722,A -85,B 0,C 180,E1 -18630,E2 -18630} C_VEL
LIN {X 0,Y 254.059,Z 388.53,A -85,B 0,C 180,E1 -18631.585,E2 -18631.585} C_VEL
LIN {X 0,Y 254.155,Z 387.943,A -85,B 0,C 180,E1 -18633.17,E2 -18633.17} C_VEL
LIN {X 0,Y 254.455,Z 385.618,A -85,B 0,C 180,E1 -18636.343,E2 -18636.343} C_VEL
LIN {X 0,Y 255.02,Z 382.746,A -85,B 0,C 180,E1 -18638.718,E2 -18638.718} C_VEL
LIN {X 0,Y 255.836,Z 378.853,A -85,B 0,C 180,E1 -18641.087,E2 -18641.087} C_VEL
LIN {X 0,Y 257.01,Z 373.828,A -85,B 0,C 180,E1 -18643.44,E2 -18643.44} C_VEL
LIN {X 0,Y 258.477,Z 367.501,A -85,B 0,C 180,E1 -18645.777,E2 -18645.777} C_VEL
LIN {X 0,Y 260.452,Z 359.579,A -85,B 0,C 180,E1 -18648.078,E2 -18648.078} C_VEL
LIN {X 0,Y 262.192,Z 351.54,A -85,B 0,C 180,E1 -18649.976,E2 -18649.976} C_VEL
LIN {X 0,Y 264.157,Z 341.656,A -85,B 0,C 180,E1 -18651.868,E2 -18651.868} C_VEL
LIN {X 0,Y 266.211,Z 330.564,A -85,B 0,C 180,E1 -18653.534,E2 -18653.534} C_VEL
LIN {X 0,Y 267.986,Z 319.688,A -85,B 0,C 180,E1 -18654.809,E2 -18654.809} C_VEL
LIN {X 0,Y 269.578,Z 307.667,A -85,B 0,C 180,E1 -18655.892,E2 -18655.892} C_VEL
LIN {X 0,Y 270.717,Z 295.31,A -85,B 0,C 180,E1 -18656.708,E2 -18656.708} C_VEL
LIN {X 0,Y 271.637,Z 282.48,A -85,B 0,C 180,E1 -18657.234,E2 -18657.234} C_VEL
LIN {X 0,Y 273.657,Z 216.347,A -85,B 0,C 180,E1 -18658.961,E2 -18658.961} C_VEL
LIN {X 0,Y 271.181,Z 208.995,A -85,B 0,C 180,E1 -18659.472,E2 -18659.472} C_VEL
LIN {X 0,Y 265.456,Z 195.254,A -85,B 0,C 180,E1 -18660.6,E2 -18660.6} C_VEL
LIN {X 0,Y 258.464,Z 180.93,A -85,B 0,C 180,E1 -18661.985,E2 -18661.985} C_VEL
LIN {X 0,Y 257.016,Z 177.764,A -85,B 0,C 180,E1 -18662.323,E2 -18662.323} C_VEL
LIN {X 0,Y 256.122,Z 174.075,A -85,B 0,C 180,E1 -18663.943,E2 -18663.943} C_VEL
LIN {X 0,Y 256.115,Z 174.08,A -85,B 0,C 180,E1 -18667.27,E2 -18667.27} C_VEL
LIN {X 0,Y 256.055,Z 174.089,A -85,B 0,C 180,E1 -18671.203,E2 -18671.203} C_VEL
LIN {X 0,Y 256.058,Z 174.086,A -85,B 0,C 180,E1 -18675.53,E2 -18675.53} C_VEL
LIN {X 0,Y 256.057,Z 174.087,A -85,B 0,C 180,E1 -18678.797,E2 -18678.797} C_VEL
LIN {X 0,Y 256.139,Z 174.074,A -85,B 0,C 180,E1 -18682.869,E2 -18682.869} C_VEL
LIN {X 0,Y 256.076,Z 174.077,A -85,B 0,C 180,E1 -18686.708,E2 -18686.708} C_VEL
LIN {X 0,Y 256.138,Z 174.073,A -85,B 0,C 180,E1 -18691.404,E2 -18691.404} C_VEL
LIN {X 0,Y 256.167,Z 174.075,A -85,B 0,C 180,E1 -18695.699,E2 -18695.699} C_VEL
LIN {X 0,Y 256.167,Z 174.069,A -85,B 0,C 180,E1 -18699.105,E2 -18699.105} C_VEL
LIN {X 0,Y 256.3,Z 174.047,A -85,B 0,C 180,E1 -18704.085,E2 -18704.085} C_VEL
LIN {X 0,Y 256.31,Z 174.058,A -85,B 0,C 180,E1 -18708.934,E2 -18708.934} C_VEL
LIN {X 0,Y 256.537,Z 174.019,A -85,B 0,C 180,E1 -18712.127,E2 -18712.127} C_VEL
LIN {X 0,Y 256.714,Z 173.997,A -85,B 0,C 180,E1 -18718.431,E2 -18718.431} C_VEL
LIN {X 0,Y 256.707,Z 173.996,A -85,B 0,C 180,E1 -18718.929,E2 -18718.929} C_VEL
LIN {X 0,Y 256.374,Z 174.041,A -85,B 0,C 180,E1 -18719.804,E2 -18719.804} C_VEL
LIN {X 0,Y 254.942,Z 174.228,A -85,B 0,C 180,E1 -18721.094,E2 -18721.094} C_VEL
LIN {X 0,Y 250.422,Z 174.789,A -85,B 0,C 180,E1 -18724.095,E2 -18724.095} C_VEL
LIN {X 0,Y 249.417,Z 174.905,A -85,B 0,C 180,E1 -18725.444,E2 -18725.444} C_VEL
LIN {X 0,Y 249.379,Z 174.907,A -85,B 0,C 180,E1 -18725.901,E2 -18725.901} C_VEL
LIN {X 0,Y 249.424,Z 174.914,A -85,B 0,C 180,E1 -18729.534,E2 -18729.534} C_VEL
LIN {X 0,Y 249.205,Z 174.938,A -85,B 0,C 180,E1 -18734.703,E2 -18734.703} C_VEL
LIN {X 0,Y 249.138,Z 174.946,A -85,B 0,C 180,E1 -18738.077,E2 -18738.077} C_VEL
LIN {X 0,Y 249.084,Z 174.955,A -85,B 0,C 180,E1 -18741.518,E2 -18741.518} C_VEL
LIN {X 0,Y 249.117,Z 174.944,A -85,B 0,C 180,E1 -18745.476,E2 -18745.476} C_VEL
LIN {X 0,Y 249.073,Z 174.957,A -85,B 0,C 180,E1 -18748.989,E2 -18748.989} C_VEL
LIN {X 0,Y 249.03,Z 174.964,A -85,B 0,C 180,E1 -18752.426,E2 -18752.426} C_VEL
LIN {X 0,Y 249.047,Z 174.962,A -85,B 0,C 180,E1 -18756.343,E2 -18756.343} C_VEL
LIN {X 0,Y 249.006,Z 174.967,A -85,B 0,C 180,E1 -18760.478,E2 -18760.478} C_VEL
LIN {X 0,Y 248.985,Z 174.967,A -85,B 0,C 180,E1 -18764.883,E2 -18764.883} C_VEL
LIN {X 0,Y 249.002,Z 174.969,A -85,B 0,C 180,E1 -18767.36,E2 -18767.36} C_VEL
LIN {X 0,Y 249.076,Z 175.059,A -85,B 0,C 180,E1 -18771.679,E2 -18771.679} C_VEL
LIN {X 0,Y 251.29,Z 183.901,A -85,B 0,C 180,E1 -18775.553,E2 -18775.553} C_VEL
LIN {X 0,Y 252.099,Z 187.493,A -85,B 0,C 180,E1 -18777.044,E2 -18777.044} C_VEL
LIN {X 0,Y 260.579,Z 206.683,A -85,B 0,C 180,E1 -18778.845,E2 -18778.845} C_VEL
LIN {X 0,Y 263.319,Z 213.694,A -85,B 0,C 180,E1 -18779.42,E2 -18779.42} C_VEL
LIN {X 0,Y 266.578,Z 234.371,A -85,B 0,C 180,E1 -18780.459,E2 -18780.459} C_VEL
LIN {X 0,Y 266.838,Z 238.331,A -85,B 0,C 180,E1 -18780.61,E2 -18780.61} C_VEL
LIN {X 0,Y 264.829,Z 296.267,A -85,B 0,C 180,E1 -18782.167,E2 -18782.167} C_VEL
LIN {X 0,Y 263.783,Z 308.633,A -85,B 0,C 180,E1 -18782.747,E2 -18782.747} C_VEL
LIN {X 0,Y 262.252,Z 321.48,A -85,B 0,C 180,E1 -18783.65,E2 -18783.65} C_VEL
LIN {X 0,Y 260.403,Z 333.683,A -85,B 0,C 180,E1 -18784.845,E2 -18784.845} C_VEL
LIN {X 0,Y 258.245,Z 345.244,A -85,B 0,C 180,E1 -18786.334,E2 -18786.334} C_VEL
LIN {X 0,Y 256.019,Z 355.656,A -85,B 0,C 180,E1 -18788.036,E2 -18788.036} C_VEL
LIN {X 0,Y 254.073,Z 364.523,A -85,B 0,C 180,E1 -18789.856,E2 -18789.856} C_VEL
LIN {X 0,Y 252.073,Z 373.404,A -85,B 0,C 180,E1 -18792.14,E2 -18792.14} C_VEL
LIN {X 0,Y 250.265,Z 380.825,A -85,B 0,C 180,E1 -18794.527,E2 -18794.527} C_VEL
LIN {X 0,Y 248.818,Z 386.785,A -85,B 0,C 180,E1 -18796.941,E2 -18796.941} C_VEL
LIN {X 0,Y 247.869,Z 391.498,A -85,B 0,C 180,E1 -18799.38,E2 -18799.38} C_VEL
LIN {X 0,Y 247.264,Z 395.1,A -85,B 0,C 180,E1 -18801.83,E2 -18801.83} C_VEL
LIN {X 0,Y 247.008,Z 396.957,A -85,B 0,C 180,E1 -18803.465,E2 -18803.465} C_VEL
LIN {X 0,Y 246.849,Z 399.347,A -85,B 0,C 180,E1 -18806.736,E2 -18806.736} C_VEL
LIN {X 0,Y 246.897,Z 399.955,A -85,B 0,C 180,E1 -18808.369,E2 -18808.369} C_VEL
LIN {X 0,Y 246.936,Z 400.167,A -85,B 0,C 180,E1 -18810,E2 -18810} C_VEL
LIN {X 0,Y 246.897,Z 399.944,A -85,B 0,C 180,E1 -18811.631,E2 -18811.631} C_VEL
LIN {X 0,Y 246.851,Z 399.33,A -85,B 0,C 180,E1 -18813.264,E2 -18813.264} C_VEL
LIN {X 0,Y 246.883,Z 398.328,A -85,B 0,C 180,E1 -18814.899,E2 -18814.899} C_VEL
LIN {X 0,Y 247.009,Z 396.924,A -85,B 0,C 180,E1 -18816.535,E2 -18816.535} C_VEL
LIN {X 0,Y 247.421,Z 393.979,A -85,B 0,C 180,E1 -18818.988,E2 -18818.988} C_VEL
LIN {X 0,Y 248.164,Z 389.997,A -85,B 0,C 180,E1 -18821.434,E2 -18821.434} C_VEL
LIN {X 0,Y 249.481,Z 383.877,A -85,B 0,C 180,E1 -18824.27,E2 -18824.27} C_VEL
LIN {X 0,Y 251.17,Z 377.199,A -85,B 0,C 180,E1 -18826.667,E2 -18826.667} C_VEL
LIN {X 0,Y 252.99,Z 369.168,A -85,B 0,C 180,E1 -18828.978,E2 -18828.978} C_VEL
LIN {X 0,Y 254.918,Z 360.411,A -85,B 0,C 180,E1 -18831.002,E2 -18831.002} C_VEL
LIN {X 0,Y 257.185,Z 349.913,A -85,B 0,C 180,E1 -18832.917,E2 -18832.917} C_VEL
LIN {X 0,Y 259.546,Z 338.096,A -85,B 0,C 180,E1 -18834.603,E2 -18834.603} C_VEL
LIN {X 0,Y 261.414,Z 326.187,A -85,B 0,C 180,E1 -18835.905,E2 -18835.905} C_VEL
LIN {X 0,Y 263.11,Z 313.792,A -85,B 0,C 180,E1 -18836.899,E2 -18836.899} C_VEL
LIN {X 0,Y 264.46,Z 301.018,A -85,B 0,C 180,E1 -18837.607,E2 -18837.607} C_VEL
LIN {X 0,Y 265.169,Z 287.477,A -85,B 0,C 180,E1 -18838.063,E2 -18838.063} C_VEL
LIN {X 0,Y 266.725,Z 235.755,A -85,B 0,C 180,E1 -18839.438,E2 -18839.438} C_VEL
LIN {X 0,Y 263.208,Z 213.377,A -85,B 0,C 180,E1 -18840.559,E2 -18840.559} C_VEL
LIN {X 0,Y 256.979,Z 198.283,A -85,B 0,C 180,E1 -18841.861,E2 -18841.861} C_VEL
LIN {X 0,Y 252.049,Z 187.407,A -85,B 0,C 180,E1 -18842.942,E2 -18842.942} C_VEL
LIN {X 0,Y 250.305,Z 179.852,A -85,B 0,C 180,E1 -18846.131,E2 -18846.131} C_VEL
LIN {X 0,Y 249.052,Z 174.963,A -85,B 0,C 180,E1 -18848.376,E2 -18848.376} C_VEL
LIN {X 0,Y 248.994,Z 174.971,A -85,B 0,C 180,E1 -18852.788,E2 -18852.788} C_VEL
LIN {X 0,Y 249.01,Z 174.966,A -85,B 0,C 180,E1 -18857.361,E2 -18857.361} C_VEL
LIN {X 0,Y 249.026,Z 174.965,A -85,B 0,C 180,E1 -18861.619,E2 -18861.619} C_VEL
LIN {X 0,Y 249.043,Z 174.963,A -85,B 0,C 180,E1 -18865.639,E2 -18865.639} C_VEL
LIN {X 0,Y 249.002,Z 174.967,A -85,B 0,C 180,E1 -18869.466,E2 -18869.466} C_VEL
LIN {X 0,Y 249.04,Z 174.958,A -85,B 0,C 180,E1 -18873.158,E2 -18873.158} C_VEL
LIN {X 0,Y 249.057,Z 174.955,A -85,B 0,C 180,E1 -18876.73,E2 -18876.73} C_VEL
LIN {X 0,Y 249.108,Z 174.954,A -85,B 0,C 180,E1 -18880.211,E2 -18880.211} C_VEL
LIN {X 0,Y 249.242,Z 174.935,A -85,B 0,C 180,E1 -18883.622,E2 -18883.622} C_VEL
LIN {X 0,Y 249.245,Z 174.932,A -85,B 0,C 180,E1 -18888.616,E2 -18888.616} C_VEL
LIN {X 0,Y 249.455,Z 174.908,A -85,B 0,C 180,E1 -18891.902,E2 -18891.902} C_VEL
LIN {X 0,Y 249.296,Z 174.928,A -85,B 0,C 180,E1 -18895.149,E2 -18895.149} C_VEL
LIN {X 0,Y 249.676,Z 174.88,A -85,B 0,C 180,E1 -18898.387,E2 -18898.387} C_VEL
LIN {X 0,Y 249.676,Z 174.884,A -85,B 0,C 180,E1 -18901.613,E2 -18901.613} C_VEL
LIN {X 0,Y 249.444,Z 174.905,A -85,B 0,C 180,E1 -18906.633,E2 -18906.633} C_VEL
